C07284=1036.536,347.439,372.467,172.361,44.359,158.643
C07285=1036.529,347.192,372.505,172.355,44.357,158.642
C07286=1036.521,346.945,372.542,172.350,44.354,158.641
C07287=1036.513,346.698,372.579,172.344,44.352,158.640
C07288=1036.505,346.451,372.616,172.339,44.349,158.638
C07289=1036.498,346.204,372.654,172.332,44.347,158.637
C07290=1036.491,345.956,372.691,172.327,44.345,158.636
C07291=1036.483,345.710,372.728,172.322,44.343,158.635
C07292=1036.475,345.462,372.766,172.316,44.340,158.634
C07293=1036.467,345.215,372.803,172.310,44.338,158.633
C07294=1036.460,344.968,372.841,172.305,44.336,158.632
C07295=1036.452,344.720,372.877,172.299,44.333,158.631
C07296=1036.445,344.473,372.914,172.294,44.331,158.630
C07297=1036.437,344.226,372.951,172.289,44.329,158.629
C07298=1036.430,343.979,372.989,172.282,44.326,158.628
C07299=1036.422,343.732,373.025,172.277,44.324,158.627
C07300=1036.415,343.485,373.063,172.272,44.322,158.626
C07301=1036.407,343.238,373.099,172.266,44.320,158.625
C07302=1036.400,342.991,373.136,172.261,44.317,158.623
C07303=1036.392,342.744,373.173,172.256,44.315,158.622
C07304=1036.385,342.497,373.210,172.249,44.313,158.621
C07305=1036.378,342.249,373.247,172.244,44.310,158.620
C07306=1036.370,342.002,373.284,172.239,44.308,158.619
C07307=1036.363,341.755,373.320,172.233,44.306,158.618
C07308=1036.355,341.508,373.358,172.228,44.303,158.617
C07309=1036.348,341.260,373.394,172.223,44.301,158.616
C07310=1036.340,341.013,373.431,172.218,44.299,158.615
C07311=1036.333,340.766,373.468,172.211,44.297,158.614
C07312=1036.325,340.518,373.504,172.206,44.295,158.613
C07313=1036.318,340.272,373.541,172.201,44.293,158.612
C07314=1036.310,340.025,373.577,172.196,44.291,158.611
C07315=1036.303,339.777,373.614,172.190,44.288,158.610
C07316=1036.295,339.530,373.651,172.185,44.286,158.609
C07317=1036.287,339.283,373.687,172.180,44.284,158.608
C07318=1036.280,339.035,373.723,172.175,44.282,158.607
C07319=1036.273,338.788,373.759,172.168,44.280,158.606
C07320=1036.265,338.541,373.796,172.163,44.278,158.605
C07321=1036.258,338.294,373.833,172.158,44.275,158.604
C07322=1036.250,338.046,373.869,172.153,44.273,158.603
C07323=1036.243,337.800,373.905,172.148,44.272,158.602
C07324=1036.236,337.552,373.941,172.142,44.270,158.601
C07325=1036.228,337.304,373.978,172.137,44.267,158.600
C07326=1036.221,337.057,374.014,172.132,44.265,158.599
C07327=1036.214,336.810,374.050,172.127,44.263,158.598
C07328=1036.206,336.563,374.087,172.121,44.261,158.597
C07329=1036.199,336.316,374.124,172.116,44.259,158.597
C07330=1036.192,336.069,374.159,172.111,44.257,158.596
C07331=1036.184,335.822,374.196,172.106,44.255,158.595
C07332=1036.176,335.574,374.232,172.101,44.253,158.594
C07333=1036.165,335.199,374.287,172.093,44.250,158.592
C07334=1036.154,334.823,374.341,172.085,44.247,158.591
C07335=1036.143,334.447,374.396,172.077,44.244,158.589
C07336=1036.132,334.071,374.450,172.070,44.241,158.588
C07337=1036.125,333.824,374.487,172.064,44.238,158.587
C07338=1036.118,333.577,374.522,172.059,44.237,158.586
C07339=1036.110,333.330,374.559,172.054,44.235,158.585
C07340=1036.103,333.082,374.594,172.049,44.233,158.584
C07341=1036.095,332.835,374.630,172.044,44.231,158.583
C07342=1036.088,332.588,374.666,172.039,44.229,158.583
C07343=1036.081,332.340,374.701,172.034,44.227,158.582
C07344=1036.073,332.093,374.738,172.029,44.226,158.581
C07345=1036.066,331.846,374.773,172.023,44.223,158.580
C07346=1036.058,331.598,374.808,172.018,44.222,158.579
C07347=1036.051,331.351,374.844,172.013,44.220,158.578
C07348=1036.044,331.103,374.880,172.008,44.218,158.577
C07349=1036.037,330.857,374.916,172.003,44.216,158.576
C07350=1036.029,330.609,374.951,171.998,44.214,158.575
C07351=1036.022,330.362,374.987,171.993,44.213,158.574
C07352=1036.015,330.114,375.022,171.988,44.210,158.573
C07353=1036.008,329.867,375.058,171.983,44.209,158.573
C07354=1036.000,329.619,375.094,171.978,44.207,158.572
C07355=1035.993,329.372,375.130,171.973,44.205,158.571
C07356=1035.986,329.124,375.165,171.968,44.203,158.570
C07357=1035.979,328.877,375.201,171.963,44.202,158.569
C07358=1035.972,328.630,375.236,171.958,44.199,158.568
C07359=1035.965,328.382,375.272,171.953,44.198,158.567
C07360=1035.957,328.136,375.307,171.948,44.196,158.567
C07361=1035.950,327.888,375.342,171.943,44.195,158.566
C07362=1035.942,327.640,375.377,171.938,44.193,158.565
C07363=1035.935,327.392,375.412,171.933,44.191,158.564
C07364=1035.927,327.145,375.447,171.928,44.189,158.563
C07365=1035.920,326.898,375.482,171.924,44.187,158.562
C07366=1035.912,326.651,375.518,171.919,44.186,158.562
C07367=1035.905,326.403,375.553,171.914,44.184,158.561
C07368=1035.897,326.156,375.588,171.909,44.183,158.560
C07369=1035.890,325.908,375.623,171.904,44.181,158.559
C07370=1035.883,325.661,375.657,171.899,44.179,158.558
C07371=1035.875,325.413,375.693,171.894,44.178,158.557
C07372=1035.868,325.166,375.727,171.890,44.176,158.557
C07373=1035.861,324.919,375.763,171.885,44.174,158.556
C07374=1035.853,324.671,375.798,171.880,44.173,158.555
C07375=1035.846,324.424,375.833,171.875,44.171,158.554
C07376=1035.839,324.177,375.867,171.870,44.169,158.553
C07377=1035.831,323.929,375.903,171.865,44.168,158.553
C07378=1035.824,323.682,375.937,171.860,44.166,158.552
C07379=1035.817,323.434,375.972,171.856,44.164,158.551
C07380=1035.810,323.186,376.006,171.851,44.163,158.550
C07381=1035.803,322.938,376.042,171.846,44.161,158.549
C07382=1035.795,322.691,376.076,171.841,44.160,158.549
C07383=1035.788,322.444,376.111,171.836,44.159,158.548
C07384=1035.781,322.197,376.146,171.832,44.157,158.547
C07385=1035.774,321.950,376.181,171.827,44.155,158.546
C07386=1035.766,321.701,376.215,171.822,44.153,158.545
C07387=1035.759,321.454,376.250,171.817,44.152,158.545
C07388=1035.752,321.207,376.285,171.813,44.150,158.544
C07389=1035.741,320.826,376.339,171.806,44.148,158.543
C07390=1035.730,320.447,376.391,171.799,44.146,158.541
C07391=1035.719,320.066,376.444,171.791,44.143,158.540
C07392=1035.709,319.685,376.498,171.785,44.141,158.539
C07393=1035.701,319.438,376.532,171.780,44.139,158.538
C07394=1035.694,319.191,376.566,171.775,44.138,158.538
C07395=1035.687,318.943,376.601,171.770,44.137,158.537
C07396=1035.680,318.696,376.636,171.766,44.135,158.536
C07397=1035.673,318.448,376.670,171.761,44.133,158.535
C07398=1035.666,318.201,376.705,171.756,44.132,158.534
C07399=1035.659,317.953,376.739,171.752,44.130,158.534
C07400=1035.652,317.706,376.774,171.747,44.129,158.533
C07401=1035.645,317.458,376.808,171.742,44.128,158.532
C07402=1035.638,317.211,376.843,171.738,44.126,158.531
C07403=1035.631,316.963,376.877,171.733,44.124,158.531
C07404=1035.624,316.716,376.912,171.729,44.123,158.530
C07405=1035.617,316.468,376.946,171.725,44.121,158.529
C07406=1035.610,316.221,376.981,171.720,44.120,158.528
C07407=1035.603,315.973,377.015,171.715,44.119,158.528
C07408=1035.596,315.725,377.049,171.711,44.117,158.527
C07409=1035.589,315.478,377.083,171.706,44.116,158.526
C07410=1035.581,315.231,377.117,171.701,44.114,158.525
C07411=1035.575,314.983,377.152,171.697,44.112,158.525
C07412=1035.567,314.736,377.186,171.692,44.111,158.524
C07413=1035.562,314.488,377.220,171.687,44.110,158.523
C07414=1035.554,314.241,377.254,171.684,44.108,158.523
C07415=1035.548,313.993,377.289,171.679,44.107,158.522
C07416=1035.540,313.746,377.323,171.675,44.106,158.521
C07417=1035.533,313.498,377.357,171.670,44.104,158.520
C07418=1035.527,313.250,377.391,171.665,44.103,158.520
C07419=1035.520,313.004,377.426,171.661,44.101,158.519
C07420=1035.513,312.756,377.460,171.657,44.100,158.518
C07421=1035.506,312.508,377.494,171.653,44.098,158.517
C07422=1035.499,312.260,377.528,171.648,44.097,158.517
C07423=1035.493,312.012,377.562,171.643,44.096,158.516
C07424=1035.486,311.765,377.595,171.639,44.094,158.515
C07425=1035.479,311.518,377.629,171.634,44.093,158.515
C07426=1035.472,311.270,377.663,171.630,44.091,158.514
C07427=1035.464,311.022,377.697,171.626,44.090,158.513
C07428=1035.457,310.775,377.731,171.621,44.089,158.513
C07429=1035.450,310.527,377.765,171.617,44.088,158.512
C07430=1035.443,310.280,377.797,171.612,44.087,158.511
C07431=1035.435,310.033,377.831,171.608,44.085,158.511
C07432=1035.428,309.785,377.865,171.604,44.084,158.510
C07433=1035.421,309.537,377.898,171.599,44.083,158.509
C07434=1035.414,309.289,377.932,171.595,44.082,158.509
C07435=1035.407,309.042,377.965,171.590,44.080,158.508
C07436=1035.400,308.795,377.999,171.586,44.079,158.507
C07437=1035.393,308.546,378.032,171.582,44.078,158.507
C07438=1035.385,308.299,378.066,171.577,44.077,158.506
C07439=1035.379,308.052,378.099,171.573,44.076,158.505
C07440=1035.371,307.804,378.132,171.568,44.075,158.505
C07441=1035.364,307.556,378.165,171.565,44.074,158.504
C07442=1035.357,307.308,378.199,171.560,44.073,158.503
C07443=1035.350,307.061,378.233,171.556,44.071,158.503
C07444=1035.343,306.813,378.266,171.551,44.070,158.502
C07445=1035.332,306.438,378.316,171.545,44.068,158.501
C07446=1035.322,306.063,378.367,171.538,44.066,158.500
C07447=1035.311,305.687,378.418,171.532,44.065,158.499
C07448=1035.300,305.312,378.467,171.526,44.063,158.498
C07449=1035.293,305.064,378.501,171.521,44.062,158.497
C07450=1035.286,304.816,378.534,171.517,44.061,158.497
C07451=1035.280,304.569,378.567,171.512,44.060,158.496
C07452=1035.272,304.321,378.601,171.509,44.058,158.496
C07453=1035.261,303.916,378.655,171.501,44.057,158.495
C07454=1035.250,303.511,378.709,171.494,44.055,158.493
C07455=1035.238,303.106,378.763,171.487,44.053,158.493
C07456=1035.227,302.701,378.817,171.481,44.051,158.492
C07457=1035.220,302.453,378.850,171.476,44.050,158.491
C07458=1035.213,302.205,378.883,171.473,44.049,158.490
C07459=1035.206,301.957,378.917,171.468,44.048,158.490
C07460=1035.199,301.710,378.949,171.464,44.047,158.489
C07461=1035.192,301.462,378.982,171.459,44.046,158.488
C07462=1035.186,301.215,379.016,171.456,44.045,158.488
C07463=1035.179,300.966,379.049,171.452,44.043,158.487
C07464=1035.172,300.719,379.081,171.447,44.043,158.487
C07465=1035.165,300.471,379.114,171.444,44.042,158.486
C07466=1035.158,300.224,379.147,171.439,44.041,158.485
C07467=1035.152,299.976,379.180,171.435,44.039,158.485
C07468=1035.144,299.728,379.213,171.430,44.038,158.484
C07469=1035.138,299.481,379.245,171.427,44.037,158.483
C07470=1035.131,299.232,379.278,171.423,44.036,158.483
C07471=1035.124,298.985,379.312,171.418,44.035,158.482
C07472=1035.117,298.737,379.344,171.415,44.034,158.482
C07473=1035.111,298.490,379.377,171.410,44.033,158.481
C07474=1035.104,298.242,379.410,171.406,44.032,158.481
C07475=1035.097,297.994,379.443,171.402,44.031,158.480
C07476=1035.090,297.747,379.475,171.398,44.030,158.479
C07477=1035.084,297.499,379.508,171.394,44.029,158.479
C07478=1035.077,297.251,379.541,171.390,44.028,158.478
C07479=1035.071,297.003,379.574,171.386,44.027,158.478
C07480=1035.064,296.756,379.606,171.382,44.026,158.477
C07481=1035.057,296.508,379.639,171.378,44.025,158.476
C07482=1035.051,296.260,379.672,171.374,44.024,158.476
C07483=1035.044,296.012,379.705,171.370,44.022,158.475
C07484=1035.037,295.764,379.737,171.366,44.022,158.475
C07485=1035.030,295.517,379.770,171.362,44.021,158.474
C07486=1035.024,295.269,379.803,171.358,44.019,158.473
C07487=1035.016,295.021,379.835,171.354,44.018,158.473
C07488=1035.010,294.774,379.868,171.350,44.018,158.472
C07489=1035.003,294.526,379.900,171.346,44.017,158.472
C07490=1034.996,294.278,379.933,171.341,44.016,158.471
C07491=1034.989,294.031,379.965,171.338,44.015,158.471
C07492=1034.983,293.783,379.997,171.334,44.014,158.470
C07493=1034.976,293.535,380.030,171.329,44.013,158.470
C07494=1034.969,293.287,380.062,171.326,44.013,158.469
C07495=1034.963,293.039,380.094,171.322,44.011,158.469
C07496=1034.956,292.792,380.126,171.318,44.011,158.468
C07497=1034.949,292.567,380.156,171.314,44.010,158.467
C07498=1034.943,292.343,380.185,171.311,44.009,158.467
C07499=1034.937,292.118,380.214,171.307,44.008,158.467
C07500=1034.930,291.894,380.243,171.304,44.008,158.466
C07501=1034.924,291.670,380.272,171.300,44.006,158.465
C07502=1034.918,291.446,380.301,171.296,44.006,158.465
C07503=1034.912,291.221,380.330,171.293,44.005,158.465
C07504=1034.906,290.997,380.360,171.289,44.005,158.464
C07505=1034.899,290.749,380.391,171.286,44.003,158.463
C07506=1034.892,290.501,380.424,171.282,44.003,158.463
C07507=1034.885,290.253,380.455,171.277,44.002,158.462
C07508=1034.879,290.005,380.488,171.274,44.001,158.462
C07509=1034.872,289.758,380.519,171.270,44.000,158.461
C07510=1034.865,289.510,380.551,171.267,43.999,158.461
C07511=1034.857,289.262,380.583,171.262,43.999,158.460
C07512=1034.851,289.014,380.616,171.259,43.998,158.460
C07513=1034.844,288.766,380.647,171.255,43.997,158.459
C07514=1034.838,288.518,380.679,171.250,43.996,158.459
C07515=1034.831,288.271,380.711,171.247,43.996,158.458
C07516=1034.823,288.022,380.743,171.243,43.994,158.458
C07517=1034.816,287.775,380.775,171.240,43.994,158.457
C07518=1034.810,287.527,380.807,171.235,43.993,158.457
C07519=1034.804,287.279,380.838,171.231,43.992,158.456
C07520=1034.797,287.032,380.870,171.228,43.991,158.456
C07521=1034.790,286.784,380.902,171.224,43.991,158.455
C07522=1034.783,286.536,380.933,171.220,43.990,158.455
C07523=1034.776,286.288,380.965,171.216,43.989,158.454
C07524=1034.769,286.040,380.997,171.213,43.988,158.454
C07525=1034.762,285.792,381.029,171.209,43.988,158.453
C07526=1034.755,285.544,381.060,171.205,43.987,158.453
C07527=1034.749,285.296,381.092,171.201,43.986,158.452
C07528=1034.742,285.048,381.123,171.197,43.985,158.452
C07529=1034.735,284.801,381.154,171.194,43.985,158.451
C07530=1034.728,284.553,381.187,171.189,43.984,158.451
C07531=1034.721,284.305,381.218,171.186,43.984,158.450
C07532=1034.714,284.057,381.250,171.182,43.983,158.450
C07533=1034.707,283.809,381.281,171.179,43.982,158.449
C07534=1034.701,283.561,381.313,171.174,43.981,158.449
C07535=1034.694,283.313,381.344,171.171,43.981,158.448
C07536=1034.687,283.065,381.376,171.167,43.980,158.448
C07537=1034.680,282.817,381.407,171.164,43.979,158.447
C07538=1034.674,282.569,381.438,171.160,43.979,158.447
C07539=1034.667,282.321,381.470,171.156,43.978,158.447
C07540=1034.660,282.074,381.501,171.152,43.978,158.446
C07541=1034.654,281.826,381.533,171.148,43.976,158.445
C07542=1034.647,281.578,381.564,171.145,43.976,158.445
C07543=1034.640,281.330,381.596,171.141,43.975,158.445
C07544=1034.633,281.082,381.627,171.137,43.975,158.444
C07545=1034.627,280.834,381.658,171.133,43.974,158.444
C07546=1034.619,280.586,381.689,171.130,43.973,158.443
C07547=1034.612,280.339,381.721,171.126,43.973,158.443
C07548=1034.606,280.090,381.751,171.123,43.972,158.442
C07549=1034.599,279.842,381.783,171.119,43.972,158.442
C07550=1034.593,279.594,381.814,171.115,43.971,158.441
C07551=1034.586,279.346,381.846,171.111,43.970,158.441
C07552=1034.579,279.098,381.877,171.108,43.970,158.440
C07553=1034.573,278.851,381.908,171.104,43.969,158.440
C07554=1034.567,278.603,381.939,171.101,43.968,158.440
C07555=1034.560,278.355,381.970,171.097,43.968,158.439
C07556=1034.553,278.107,382.002,171.094,43.967,158.439
C07557=1034.544,277.761,382.045,171.088,43.966,158.438
C07558=1034.534,277.414,382.088,171.083,43.965,158.437
C07559=1034.524,277.067,382.131,171.078,43.965,158.437
C07560=1034.515,276.721,382.175,171.073,43.964,158.436
C07561=1034.508,276.473,382.206,171.070,43.963,158.436
C07562=1034.501,276.224,382.237,171.066,43.963,158.435
C07563=1034.494,275.977,382.268,171.063,43.962,158.435
C07564=1034.488,275.728,382.299,171.058,43.962,158.434
C07565=1034.481,275.480,382.330,171.055,43.961,158.434
C07566=1034.475,275.233,382.360,171.051,43.961,158.434
C07567=1034.468,274.985,382.391,171.048,43.960,158.433
C07568=1034.461,274.737,382.423,171.044,43.960,158.433
C07569=1034.454,274.489,382.453,171.041,43.959,158.432
C07570=1034.447,274.241,382.484,171.037,43.958,158.432
C07571=1034.441,273.992,382.515,171.034,43.958,158.431
C07572=1034.435,273.745,382.545,171.030,43.957,158.431
C07573=1034.427,273.497,382.576,171.027,43.957,158.431
C07574=1034.421,273.249,382.607,171.023,43.956,158.430
C07575=1034.413,273.001,382.638,171.019,43.956,158.430
C07576=1034.407,272.752,382.668,171.016,43.955,158.429
C07577=1034.400,272.505,382.700,171.012,43.955,158.429
C07578=1034.394,272.257,382.729,171.009,43.954,158.428
C07579=1034.387,272.009,382.760,171.005,43.954,158.428
C07580=1034.380,271.761,382.791,171.002,43.953,158.428
C07581=1034.373,271.512,382.822,170.998,43.953,158.427
C07582=1034.368,271.265,382.852,170.995,43.953,158.427
C07583=1034.360,271.017,382.883,170.992,43.952,158.426
C07584=1034.354,270.768,382.914,170.988,43.951,158.426
C07585=1034.347,270.520,382.944,170.985,43.951,158.425
C07586=1034.341,270.272,382.974,170.981,43.951,158.425
C07587=1034.333,270.025,383.005,170.978,43.950,158.425
C07588=1034.326,269.777,383.035,170.973,43.949,158.424
C07589=1034.320,269.528,383.066,170.970,43.949,158.424
C07590=1034.313,269.281,383.096,170.967,43.949,158.423
C07591=1034.307,269.032,383.126,170.963,43.948,158.423
C07592=1034.299,268.784,383.157,170.960,43.948,158.423
C07593=1034.293,268.536,383.188,170.956,43.947,158.422
C07594=1034.286,268.288,383.218,170.953,43.947,158.422
C07595=1034.279,268.040,383.248,170.950,43.947,158.422
C07596=1034.273,267.792,383.278,170.946,43.946,158.421
C07597=1034.266,267.544,383.308,170.943,43.945,158.421
C07598=1034.260,267.296,383.339,170.939,43.945,158.420
C07599=1034.253,267.047,383.369,170.936,43.945,158.420
C07600=1034.246,266.800,383.400,170.932,43.945,158.420
C07601=1034.239,266.552,383.430,170.929,43.944,158.419
C07602=1034.232,266.304,383.460,170.926,43.943,158.419
C07603=1034.225,266.056,383.490,170.922,43.943,158.418
C07604=1034.219,265.807,383.520,170.919,43.943,158.418
C07605=1034.212,265.559,383.550,170.915,43.943,158.418
C07606=1034.205,265.311,383.580,170.912,43.942,158.417
C07607=1034.199,265.063,383.610,170.909,43.942,158.417
C07608=1034.192,264.815,383.641,170.905,43.941,158.416
C07609=1034.186,264.567,383.671,170.902,43.941,158.416
C07610=1034.178,264.319,383.701,170.898,43.941,158.416
C07611=1034.172,264.070,383.731,170.895,43.941,158.415
C07612=1034.165,263.823,383.761,170.892,43.940,158.415
C07613=1034.156,263.481,383.803,170.887,43.939,158.415
C07614=1034.147,263.139,383.844,170.883,43.939,158.414
C07615=1034.138,262.798,383.885,170.878,43.939,158.414
C07616=1034.129,262.455,383.926,170.874,43.938,158.413
C07617=1034.122,262.207,383.956,170.870,43.937,158.413
C07618=1034.115,261.959,383.986,170.867,43.937,158.412
C07619=1034.109,261.711,384.017,170.863,43.937,158.412
C07620=1034.102,261.463,384.047,170.860,43.937,158.412
C07621=1034.095,261.215,384.076,170.857,43.936,158.411
C07622=1034.088,260.966,384.106,170.853,43.936,158.411
C07623=1034.081,260.718,384.135,170.850,43.936,158.411
C07624=1034.074,260.470,384.165,170.847,43.935,158.410
C07625=1034.067,260.222,384.195,170.843,43.935,158.410
C07626=1034.061,259.974,384.224,170.840,43.935,158.409
C07627=1034.053,259.726,384.254,170.837,43.935,158.409
C07628=1034.047,259.478,384.283,170.833,43.935,158.409
C07629=1034.040,259.229,384.313,170.830,43.935,158.408
C07630=1034.033,258.981,384.342,170.827,43.934,158.408
C07631=1034.026,258.733,384.372,170.823,43.934,158.408
C07632=1034.019,258.484,384.401,170.820,43.934,158.407
C07633=1034.013,258.237,384.431,170.817,43.934,158.407
C07634=1034.006,257.988,384.460,170.813,43.933,158.407
C07635=1033.999,257.741,384.490,170.810,43.933,158.406
C07636=1033.992,257.492,384.519,170.807,43.933,158.406
C07637=1033.986,257.244,384.549,170.803,43.933,158.406
C07638=1033.979,256.995,384.579,170.800,43.932,158.405
C07639=1033.972,256.748,384.608,170.797,43.932,158.405
C07640=1033.965,256.499,384.637,170.793,43.932,158.405
C07641=1033.958,256.251,384.666,170.790,43.932,158.404
C07642=1033.951,256.003,384.696,170.788,43.931,158.404
C07643=1033.945,255.755,384.725,170.784,43.931,158.404
C07644=1033.938,255.507,384.755,170.781,43.931,158.404
C07645=1033.932,255.259,384.784,170.778,43.931,158.403
C07646=1033.924,255.010,384.813,170.774,43.931,158.403
C07647=1033.917,254.763,384.843,170.771,43.931,158.402
C07648=1033.911,254.514,384.872,170.768,43.930,158.402
C07649=1033.904,254.266,384.901,170.765,43.930,158.402
C07650=1033.898,254.018,384.931,170.761,43.930,158.401
C07651=1033.891,253.769,384.961,170.758,43.930,158.401
C07652=1033.884,253.521,384.989,170.755,43.930,158.401
C07653=1033.877,253.273,385.018,170.752,43.929,158.401
C07654=1033.871,253.025,385.048,170.749,43.929,158.400
C07655=1033.864,252.776,385.078,170.746,43.929,158.400
C07656=1033.857,252.528,385.107,170.742,43.929,158.400
C07657=1033.851,252.280,385.136,170.739,43.929,158.399
C07658=1033.843,252.032,385.165,170.736,43.929,158.399
C07659=1033.837,251.784,385.194,170.732,43.928,158.399
C07660=1033.831,251.536,385.223,170.730,43.928,158.398
C07661=1033.824,251.287,385.253,170.727,43.928,158.398
C07662=1033.818,251.039,385.282,170.723,43.928,158.398
C07663=1033.811,250.791,385.312,170.720,43.928,158.397
C07664=1033.804,250.543,385.340,170.717,43.927,158.397
C07665=1033.797,250.295,385.369,170.713,43.927,158.397
C07666=1033.791,250.047,385.398,170.710,43.927,158.396
C07667=1033.784,249.798,385.428,170.708,43.927,158.396
C07668=1033.778,249.550,385.457,170.705,43.927,158.396
C07669=1033.768,249.207,385.498,170.700,43.926,158.395
C07670=1033.760,248.864,385.538,170.696,43.926,158.395
C07671=1033.750,248.520,385.578,170.691,43.926,158.395
C07672=1033.741,248.177,385.618,170.687,43.925,158.394
C07673=1033.735,247.929,385.647,170.684,43.925,158.394
C07674=1033.728,247.680,385.676,170.681,43.925,158.394
C07675=1033.722,247.432,385.705,170.678,43.925,158.393
C07676=1033.715,247.184,385.734,170.675,43.925,158.393
C07677=1033.709,246.936,385.763,170.671,43.924,158.392
C07678=1033.702,246.687,385.792,170.668,43.924,158.392
C07679=1033.696,246.439,385.821,170.666,43.924,158.392
C07680=1033.689,246.191,385.850,170.663,43.924,158.392
C07681=1033.682,245.943,385.879,170.659,43.924,158.391
C07682=1033.676,245.694,385.908,170.656,43.924,158.391
C07683=1033.669,245.446,385.937,170.654,43.924,158.391
C07684=1033.663,245.198,385.966,170.650,43.923,158.390
C07685=1033.657,244.950,385.995,170.647,43.923,158.390
C07686=1033.650,244.702,386.024,170.644,43.923,158.390
C07687=1033.643,244.452,386.052,170.641,43.923,158.390
C07688=1033.637,244.204,386.081,170.638,43.923,158.389
C07689=1033.630,243.956,386.110,170.635,43.923,158.389
C07690=1033.624,243.708,386.139,170.632,43.923,158.389
C07691=1033.617,243.461,386.167,170.628,43.923,158.388
C07692=1033.610,243.211,386.196,170.626,43.922,158.388
C07693=1033.603,242.963,386.224,170.623,43.922,158.388
C07694=1033.597,242.715,386.253,170.620,43.922,158.388
C07695=1033.590,242.467,386.282,170.616,43.922,158.387
C07696=1033.584,242.219,386.310,170.614,43.922,158.387
C07697=1033.577,241.970,386.339,170.611,43.922,158.387
C07698=1033.570,241.722,386.368,170.608,43.922,158.386
C07699=1033.564,241.473,386.396,170.604,43.922,158.386
C07700=1033.557,241.225,386.425,170.602,43.922,158.386
C07701=1033.550,240.977,386.453,170.599,43.922,158.386
C07702=1033.544,240.729,386.482,170.596,43.922,158.385
C07703=1033.537,240.481,386.510,170.592,43.921,158.385
C07704=1033.531,240.232,386.539,170.590,43.921,158.385
C07705=1033.524,239.984,386.567,170.587,43.921,158.384
C07706=1033.517,239.736,386.596,170.583,43.921,158.384
C07707=1033.511,239.487,386.624,170.580,43.922,158.384
C07708=1033.504,239.239,386.652,170.578,43.922,158.384
C07709=1033.497,238.991,386.680,170.575,43.921,158.383
C07710=1033.490,238.742,386.710,170.572,43.921,158.383
C07711=1033.484,238.494,386.737,170.568,43.921,158.383
C07712=1033.477,238.246,386.766,170.566,43.921,158.383
C07713=1033.470,237.997,386.793,170.563,43.921,158.382
C07714=1033.464,237.749,386.823,170.560,43.921,158.382
C07715=1033.457,237.501,386.850,170.557,43.922,158.382
C07716=1033.450,237.253,386.879,170.554,43.921,158.382
C07717=1033.443,237.004,386.906,170.551,43.921,158.381
C07718=1033.438,236.756,386.935,170.548,43.921,158.381
C07719=1033.430,236.507,386.964,170.544,43.921,158.381
C07720=1033.423,236.259,386.991,170.542,43.921,158.381
C07721=1033.416,236.011,387.020,170.539,43.922,158.380
C07722=1033.410,235.762,387.047,170.536,43.922,158.380
C07723=1033.404,235.514,387.076,170.534,43.921,158.380
C07724=1033.397,235.266,387.104,170.530,43.921,158.380
C07725=1033.387,234.916,387.144,170.526,43.921,158.379
C07726=1033.378,234.568,387.183,170.522,43.922,158.379
C07727=1033.368,234.218,387.222,170.519,43.922,158.379
C07728=1033.359,233.869,387.262,170.514,43.922,158.378
C07729=1033.352,233.620,387.290,170.511,43.922,158.378
C07730=1033.346,233.372,387.318,170.508,43.922,158.378
C07731=1033.339,233.123,387.346,170.506,43.921,158.377
C07732=1033.332,232.875,387.374,170.502,43.921,158.377
C07733=1033.326,232.627,387.402,170.499,43.922,158.377
C07734=1033.319,232.378,387.430,170.497,43.922,158.377
C07735=1033.313,232.130,387.458,170.494,43.922,158.376
C07736=1033.306,231.882,387.487,170.490,43.922,158.376
C07737=1033.299,231.633,387.514,170.488,43.922,158.376
C07738=1033.293,231.385,387.542,170.485,43.922,158.376
C07739=1033.286,231.137,387.570,170.482,43.922,158.376
C07740=1033.279,230.888,387.598,170.480,43.922,158.375
C07741=1033.273,230.640,387.625,170.477,43.922,158.375
C07742=1033.267,230.392,387.653,170.473,43.922,158.375
C07743=1033.260,230.144,387.681,170.471,43.922,158.375
C07744=1033.253,229.896,387.709,170.468,43.922,158.374
C07745=1033.246,229.647,387.737,170.465,43.922,158.374
C07746=1033.240,229.399,387.764,170.463,43.922,158.374
C07747=1033.233,229.150,387.792,170.459,43.922,158.374
C07748=1033.227,228.902,387.820,170.456,43.923,158.373
C07749=1033.220,228.653,387.848,170.454,43.923,158.373
C07750=1033.214,228.405,387.876,170.451,43.923,158.373
C07751=1033.207,228.156,387.904,170.448,43.922,158.373
C07752=1033.200,227.908,387.931,170.445,43.923,158.373
C07753=1033.193,227.660,387.958,170.442,43.923,158.372
C07754=1033.186,227.411,387.986,170.440,43.923,158.372
C07755=1033.179,227.163,388.014,170.437,43.923,158.372
C07756=1033.173,226.914,388.042,170.434,43.923,158.372
C07757=1033.166,226.666,388.069,170.432,43.923,158.371
C07758=1033.160,226.417,388.096,170.428,43.923,158.371
C07759=1033.153,226.169,388.123,170.425,43.923,158.371
C07760=1033.146,225.921,388.151,170.423,43.924,158.371
C07761=1033.140,225.673,388.179,170.420,43.924,158.371
C07762=1033.133,225.424,388.206,170.418,43.924,158.370
C07763=1033.126,225.176,388.234,170.414,43.924,158.370
C07764=1033.119,224.928,388.261,170.411,43.925,158.370
C07765=1033.112,224.679,388.288,170.409,43.924,158.370
C07766=1033.106,224.430,388.316,170.406,43.924,158.369
C07767=1033.099,224.182,388.344,170.403,43.925,158.369
C07768=1033.092,223.933,388.371,170.401,43.925,158.369
C07769=1033.086,223.686,388.398,170.398,43.925,158.369
C07770=1033.079,223.437,388.425,170.395,43.925,158.369
C07771=1033.072,223.188,388.453,170.392,43.925,158.368
C07772=1033.066,222.940,388.481,170.389,43.926,158.368
C07773=1033.059,222.691,388.508,170.387,43.925,158.368
C07774=1033.052,222.443,388.535,170.384,43.926,158.368
C07775=1033.045,222.194,388.562,170.381,43.926,158.368
C07776=1033.039,221.946,388.590,170.378,43.926,158.367
C07777=1033.033,221.697,388.617,170.375,43.926,158.367
C07778=1033.025,221.449,388.644,170.373,43.926,158.367
C07779=1033.019,221.201,388.672,170.370,43.927,158.367
C07780=1033.012,220.952,388.699,170.368,43.926,158.367
C07781=1033.003,220.596,388.739,170.363,43.926,158.366
C07782=1032.993,220.239,388.778,170.359,43.927,158.366
C07783=1032.984,219.883,388.817,170.356,43.927,158.366
C07784=1032.975,219.526,388.856,170.352,43.927,158.365
C07785=1032.968,219.277,388.882,170.348,43.927,158.365
C07786=1032.961,219.028,388.910,170.346,43.928,158.365
C07787=1032.954,218.780,388.936,170.343,43.928,158.365
C07788=1032.947,218.531,388.964,170.341,43.928,158.365
C07789=1032.941,218.283,388.990,170.338,43.929,158.364
C07790=1032.934,218.035,389.018,170.336,43.928,158.364
C07791=1032.927,217.786,389.044,170.333,43.929,158.364
C07792=1032.920,217.538,389.072,170.330,43.929,158.364
C07793=1032.913,217.289,389.098,170.328,43.929,158.364
C07794=1032.907,217.041,389.126,170.324,43.929,158.363
C07795=1032.900,216.792,389.152,170.322,43.930,158.363
C07796=1032.893,216.544,389.180,170.319,43.930,158.363
C07797=1032.886,216.295,389.206,170.317,43.930,158.363
C07798=1032.880,216.047,389.234,170.314,43.931,158.363
C07799=1032.873,215.799,389.260,170.312,43.930,158.363
C07800=1032.867,215.550,389.287,170.309,43.931,158.362
C07801=1032.859,215.301,389.314,170.306,43.931,158.362
C07802=1032.854,215.053,389.341,170.303,43.931,158.362
C07803=1032.846,214.805,389.368,170.300,43.932,158.362
C07804=1032.840,214.556,389.395,170.298,43.932,158.362
C07805=1032.833,214.308,389.421,170.295,43.932,158.361
C07806=1032.827,214.059,389.449,170.293,43.932,158.361
C07807=1032.819,213.811,389.475,170.290,43.933,158.361
C07808=1032.813,213.562,389.502,170.287,43.932,158.361
C07809=1032.806,213.314,389.529,170.284,43.933,158.361
C07810=1032.800,213.065,389.556,170.282,43.933,158.360
C07811=1032.793,212.816,389.582,170.279,43.933,158.360
C07812=1032.787,212.569,389.610,170.277,43.934,158.360
C07813=1032.780,212.320,389.636,170.274,43.934,158.360
C07814=1032.773,212.071,389.663,170.272,43.934,158.360
C07815=1032.767,211.823,389.689,170.268,43.934,158.360
C07816=1032.760,211.574,389.717,170.266,43.934,158.359
C07817=1032.753,211.326,389.743,170.263,43.934,158.359
C07818=1032.747,211.077,389.770,170.261,43.935,158.359
C07819=1032.740,210.828,389.797,170.258,43.935,158.359
C07820=1032.733,210.580,389.823,170.256,43.935,158.359
C07821=1032.727,210.332,389.850,170.253,43.936,158.359
C07822=1032.720,210.083,389.877,170.251,43.936,158.358
C07823=1032.713,209.835,389.903,170.248,43.936,158.358
C07824=1032.707,209.586,389.930,170.246,43.936,158.358
C07825=1032.700,209.337,389.956,170.242,43.937,158.358
C07826=1032.693,209.089,389.982,170.240,43.937,158.358
C07827=1032.687,208.840,390.009,170.237,43.937,158.358
C07828=1032.680,208.593,390.036,170.235,43.938,158.357
C07829=1032.673,208.344,390.062,170.233,43.937,158.357
C07830=1032.666,208.095,390.089,170.230,43.938,158.357
C07831=1032.660,207.847,390.116,170.228,43.938,158.357
C07832=1032.653,207.598,390.142,170.225,43.938,158.357
C07833=1032.646,207.350,390.168,170.223,43.939,158.357
C07834=1032.639,207.101,390.194,170.220,43.939,158.356
C07835=1032.632,206.853,390.221,170.217,43.939,158.356
C07836=1032.626,206.604,390.248,170.214,43.940,158.356
C07837=1032.617,206.253,390.284,170.211,43.940,158.356
C07838=1032.606,205.902,390.322,170.207,43.940,158.356
C07839=1032.597,205.551,390.359,170.204,43.941,158.355
C07840=1032.588,205.200,390.396,170.200,43.942,158.355
C07841=1032.562,204.151,390.501,169.861,43.837,158.304
C07842=1032.556,203.902,390.527,169.857,43.838,158.304
C07843=1032.550,203.653,390.551,169.853,43.839,158.304
C07844=1032.544,203.405,390.576,169.850,43.840,158.304
C07845=1032.537,203.157,390.601,169.846,43.842,158.304
C07846=1032.531,202.907,390.626,169.842,43.842,158.304
C07847=1032.525,202.659,390.651,169.839,43.844,158.304
C07848=1032.519,202.411,390.676,169.835,43.844,158.304
C07849=1032.514,202.161,390.701,169.832,43.846,158.304
C07850=1032.507,201.913,390.726,169.828,43.847,158.304
C07851=1032.501,201.664,390.751,169.825,43.848,158.303
C07852=1032.495,201.416,390.775,169.822,43.849,158.303
C07853=1032.489,201.167,390.800,169.817,43.850,158.303
C07854=1032.483,200.918,390.825,169.815,43.851,158.303
C07855=1032.477,200.669,390.850,169.811,43.852,158.303
C07856=1032.472,200.421,390.875,169.808,43.853,158.303
C07857=1032.465,200.172,390.899,169.804,43.854,158.303
C07858=1032.459,199.923,390.924,169.800,43.856,158.303
C07859=1032.452,199.675,390.949,169.797,43.857,158.303
C07860=1032.446,199.426,390.973,169.794,43.858,158.303
C07861=1032.440,199.177,390.997,169.790,43.859,158.303
C07862=1032.434,198.928,391.022,169.787,43.860,158.303
C07863=1032.427,198.679,391.046,169.783,43.862,158.303
C07864=1032.422,198.431,391.071,169.780,43.863,158.303
C07865=1032.415,198.182,391.095,169.776,43.865,158.303
C07866=1032.409,197.933,391.120,169.773,43.865,158.302
C07867=1032.403,197.685,391.144,169.769,43.867,158.302
C07868=1032.397,197.436,391.169,169.765,43.868,158.302
C07869=1032.390,197.187,391.193,169.763,43.869,158.302
C07870=1032.384,196.938,391.218,169.759,43.871,158.302
C07871=1032.378,196.690,391.242,169.756,43.872,158.302
C07872=1032.372,196.441,391.267,169.752,43.873,158.302
C07873=1032.365,196.192,391.291,169.749,43.874,158.302
C07874=1032.360,195.943,391.315,169.745,43.875,158.302
C07875=1032.353,195.695,391.340,169.741,43.877,158.302
C07876=1032.348,195.446,391.364,169.739,43.878,158.302
C07877=1032.341,195.197,391.388,169.735,43.879,158.302
C07878=1032.335,194.948,391.413,169.732,43.880,158.302
C07879=1032.329,194.701,391.437,169.728,43.882,158.302
C07880=1032.323,194.451,391.462,169.725,43.882,158.302
C07881=1032.316,194.202,391.486,169.721,43.884,158.302
C07882=1032.311,193.954,391.510,169.719,43.885,158.302
C07883=1032.304,193.705,391.534,169.715,43.886,158.302
C07884=1032.299,193.456,391.558,169.712,43.888,158.302
C07885=1032.292,193.208,391.583,169.708,43.889,158.302
C07886=1032.287,192.959,391.607,169.705,43.890,158.302
C07887=1032.280,192.710,391.631,169.701,43.892,158.302
C07888=1032.274,192.461,391.656,169.699,43.893,158.302
C07889=1032.268,192.213,391.679,169.695,43.894,158.302
C07890=1032.262,191.963,391.704,169.692,43.895,158.302
C07891=1032.256,191.715,391.728,169.688,43.896,158.302
C07892=1032.250,191.466,391.752,169.685,43.898,158.302
C07893=1032.244,191.217,391.776,169.681,43.899,158.301
C07894=1032.238,190.968,391.801,169.678,43.900,158.301
C07895=1032.232,190.720,391.824,169.675,43.902,158.301
C07896=1032.226,190.471,391.849,169.672,43.903,158.301
C07897=1032.220,190.222,391.873,169.668,43.904,158.301
C07898=1032.214,189.973,391.897,169.665,43.906,158.301
C07899=1032.208,189.725,391.921,169.661,43.907,158.301
C07900=1032.202,189.476,391.945,169.658,43.908,158.301
C07901=1032.196,189.227,391.969,169.656,43.909,158.301
C07902=1032.190,188.944,391.997,169.652,43.911,158.301
C07903=1032.183,188.660,392.024,169.648,43.912,158.301
C07904=1032.176,188.376,392.051,169.644,43.914,158.301
C07905=1032.169,188.093,392.079,169.640,43.915,158.301
C07906=1032.163,187.844,392.103,169.637,43.916,158.301
C07907=1032.157,187.595,392.127,169.634,43.918,158.301
C07908=1032.151,187.346,392.152,169.631,43.919,158.301
C07909=1032.145,187.098,392.175,169.627,43.920,158.301
C07910=1032.140,186.849,392.199,169.624,43.922,158.301
C07911=1032.134,186.600,392.223,169.620,43.923,158.301
C07912=1032.127,186.351,392.246,169.618,43.924,158.301
C07913=1032.122,186.102,392.271,169.615,43.925,158.301
C07914=1032.116,185.854,392.295,169.611,43.927,158.301
C07915=1032.110,185.605,392.319,169.608,43.928,158.301
C07916=1032.104,185.355,392.342,169.604,43.930,158.301
C07917=1032.099,185.107,392.367,169.601,43.931,158.301
C07918=1032.093,184.859,392.390,169.599,43.932,158.301
C07919=1032.086,184.610,392.414,169.595,43.933,158.301
C07920=1032.081,184.361,392.438,169.592,43.935,158.301
C07921=1032.074,184.111,392.462,169.588,43.936,158.301
C07922=1032.069,183.863,392.486,169.585,43.937,158.301
C07923=1032.063,183.615,392.510,169.583,43.938,158.301
C07924=1032.058,183.366,392.534,169.579,43.940,158.301
C07925=1032.051,183.116,392.557,169.576,43.941,158.301
C07926=1032.045,182.868,392.581,169.573,43.942,158.301
C07927=1032.039,182.619,392.604,169.569,43.944,158.301
C07928=1032.033,182.370,392.628,169.566,43.945,158.301
C07929=1032.027,182.121,392.651,169.563,43.947,158.301
C07930=1032.020,181.873,392.674,169.560,43.948,158.301
C07931=1032.014,181.624,392.697,169.556,43.950,158.301
C07932=1032.007,181.375,392.721,169.554,43.952,158.301
C07933=1032.002,181.126,392.744,169.550,43.953,158.301
C07934=1031.996,180.878,392.768,169.547,43.954,158.301
C07935=1031.989,180.628,392.791,169.544,43.956,158.301
C07936=1031.983,180.380,392.815,169.541,43.958,158.301
C07937=1031.977,180.131,392.837,169.538,43.959,158.301
C07938=1031.971,179.882,392.860,169.534,43.961,158.301
C07939=1031.964,179.633,392.884,169.531,43.962,158.301
C07940=1031.959,179.384,392.907,169.528,43.963,158.301
C07941=1031.952,179.135,392.931,169.525,43.965,158.301
C07942=1031.946,178.887,392.954,169.522,43.967,158.301
C07943=1031.940,178.638,392.976,169.518,43.968,158.301
C07944=1031.933,178.389,393.000,169.516,43.970,158.302
C07945=1031.928,178.140,393.023,169.513,43.971,158.302
C07946=1031.922,177.891,393.046,169.509,43.973,158.301
C07947=1031.915,177.642,393.070,169.506,43.974,158.302
C07948=1031.909,177.394,393.093,169.503,43.976,158.302
C07949=1031.903,177.145,393.116,169.500,43.977,158.302
C07950=1031.897,176.896,393.139,169.497,43.979,158.302
C07951=1031.891,176.647,393.163,169.493,43.980,158.302
C07952=1031.885,176.398,393.186,169.491,43.982,158.302
C07953=1031.879,176.149,393.209,169.488,43.983,158.302
C07954=1031.872,175.900,393.232,169.484,43.985,158.302
C07955=1031.866,175.651,393.255,169.481,43.986,158.302
C07956=1031.860,175.403,393.278,169.478,43.988,158.302
C07957=1031.855,175.154,393.301,169.475,43.989,158.302
C07958=1031.849,174.905,393.324,169.472,43.991,158.302
C07959=1031.841,174.656,393.347,169.468,43.993,158.302
C07960=1031.836,174.407,393.370,169.466,43.994,158.302
C07961=1031.830,174.158,393.393,169.463,43.996,158.302
C07962=1031.824,173.909,393.416,169.459,43.997,158.302
C07963=1031.818,173.660,393.440,169.456,43.999,158.302
C07964=1031.811,173.412,393.462,169.454,44.000,158.302
C07965=1031.805,173.163,393.485,169.450,44.002,158.302
C07966=1031.799,172.879,393.511,169.447,44.004,158.302
C07967=1031.792,172.594,393.538,169.444,44.005,158.302
C07968=1031.785,172.311,393.564,169.440,44.007,158.302
C07969=1031.778,172.026,393.590,169.436,44.009,158.302
C07970=1031.772,171.777,393.613,169.434,44.011,158.303
C07971=1031.767,171.528,393.636,169.431,44.012,158.303
C07972=1031.760,171.280,393.659,169.427,44.014,158.303
C07973=1031.754,171.031,393.682,169.424,44.015,158.303
C07974=1031.748,170.783,393.705,169.422,44.016,158.303
C07975=1031.742,170.533,393.728,169.419,44.018,158.303
C07976=1031.736,170.284,393.751,169.415,44.020,158.303
C07977=1031.730,170.035,393.774,169.413,44.021,158.303
C07978=1031.724,169.787,393.796,169.410,44.023,158.303
C07979=1031.718,169.538,393.819,169.407,44.024,158.303
C07980=1031.713,169.289,393.842,169.403,44.026,158.303
C07981=1031.706,169.040,393.865,169.400,44.027,158.303
C07982=1031.700,168.791,393.888,169.398,44.029,158.303
C07983=1031.695,168.542,393.911,169.394,44.031,158.303
C07984=1031.689,168.294,393.934,169.391,44.032,158.303
C07985=1031.683,168.045,393.957,169.389,44.034,158.303
C07986=1031.677,167.796,393.979,169.386,44.035,158.303
C07987=1031.671,167.547,394.002,169.383,44.036,158.303
C07988=1031.665,167.298,394.025,169.379,44.038,158.303
C07989=1031.659,167.049,394.048,169.377,44.039,158.303
C07990=1031.652,166.800,394.070,169.374,44.041,158.303
C07991=1031.647,166.551,394.093,169.371,44.043,158.303
C07992=1031.641,166.302,394.116,169.367,44.044,158.303
C07993=1031.636,166.053,394.139,169.365,44.046,158.304
C07994=1031.629,165.804,394.161,169.362,44.047,158.304
C07995=1031.623,165.555,394.184,169.359,44.049,158.304
C07996=1031.618,165.306,394.207,169.357,44.050,158.304
C07997=1031.612,165.057,394.230,169.353,44.052,158.304
C07998=1031.605,164.809,394.252,169.350,44.054,158.304
C07999=1031.600,164.559,394.274,169.347,44.055,158.304
C08000=1031.594,164.310,394.297,169.345,44.057,158.304
C08001=1031.589,164.062,394.320,169.342,44.058,158.304
C08002=1031.583,163.814,394.342,169.338,44.060,158.304
C08003=1031.577,163.565,394.365,169.335,44.061,158.304
C08004=1031.571,163.316,394.388,169.333,44.063,158.304
C08005=1031.566,163.066,394.410,169.330,44.064,158.304
C08006=1031.559,162.818,394.433,169.327,44.066,158.304
C08007=1031.554,162.569,394.456,169.324,44.068,158.304
C08008=1031.548,162.320,394.479,169.321,44.069,158.304
C08009=1031.542,162.070,394.501,169.318,44.070,158.304
C08010=1031.536,161.822,394.523,169.315,44.072,158.304
C08011=1031.530,161.573,394.546,169.313,44.073,158.304
C08012=1031.525,161.324,394.569,169.310,44.075,158.305
C08013=1031.519,161.075,394.591,169.306,44.077,158.305
C08014=1031.513,160.826,394.614,169.304,44.079,158.305
C08015=1031.508,160.578,394.636,169.301,44.080,158.305
C08016=1031.502,160.328,394.658,169.298,44.081,158.305
C08017=1031.496,160.080,394.681,169.295,44.083,158.305
C08018=1031.490,159.831,394.704,169.293,44.084,158.305
C08019=1031.484,159.581,394.726,169.290,44.086,158.305
C08020=1031.478,159.333,394.748,169.286,44.087,158.305
C08021=1031.472,159.084,394.770,169.284,44.089,158.305
C08022=1031.466,158.835,394.793,169.281,44.091,158.305
C08023=1031.460,158.585,394.815,169.278,44.093,158.305
C08024=1031.453,158.337,394.837,169.276,44.094,158.305
C08025=1031.448,158.087,394.859,169.272,44.096,158.306
C08026=1031.442,157.839,394.881,169.269,44.098,158.306
C08027=1031.436,157.590,394.903,169.267,44.100,158.306
C08028=1031.430,157.341,394.926,169.264,44.101,158.306
C08029=1031.424,157.092,394.947,169.261,44.103,158.306
C08030=1031.417,156.808,394.973,169.258,44.105,158.306
C08031=1031.410,156.523,394.997,169.254,44.107,158.306
C08032=1031.403,156.238,395.023,169.251,44.109,158.306
C08033=1031.396,155.954,395.049,169.248,44.111,158.306
C08034=1031.390,155.705,395.070,169.245,44.112,158.306
C08035=1031.385,155.455,395.093,169.242,44.114,158.306
C08036=1031.379,155.207,395.115,169.240,44.116,158.307
C08037=1031.373,154.958,395.136,169.236,44.117,158.306
C08038=1031.366,154.710,395.159,169.233,44.119,158.307
C08039=1031.361,154.460,395.181,169.231,44.121,158.307
C08040=1031.354,154.211,395.202,169.228,44.122,158.307
C08041=1031.348,153.962,395.225,169.225,44.124,158.307
C08042=1031.343,153.713,395.247,169.223,44.126,158.307
C08043=1031.337,153.464,395.268,169.220,44.127,158.307
C08044=1031.331,153.215,395.290,169.216,44.130,158.307
C08045=1031.324,152.966,395.312,169.214,44.131,158.307
C08046=1031.318,152.717,395.334,169.211,44.133,158.307
C08047=1031.312,152.468,395.356,169.208,44.135,158.307
C08048=1031.307,152.220,395.377,169.206,44.136,158.308
C08049=1031.301,151.971,395.400,169.203,44.138,158.308
C08050=1031.295,151.721,395.421,169.199,44.140,158.308
C08051=1031.288,151.472,395.443,169.197,44.142,158.308
C08052=1031.282,151.223,395.465,169.194,44.144,158.308
C08053=1031.276,150.975,395.487,169.191,44.145,158.308
C08054=1031.270,150.726,395.508,169.189,44.147,158.308
C08055=1031.264,150.477,395.530,169.186,44.149,158.308
C08056=1031.259,150.227,395.552,169.184,44.151,158.308
C08057=1031.253,149.978,395.574,169.181,44.152,158.308
C08058=1031.247,149.730,395.595,169.177,44.154,158.308
C08059=1031.240,149.481,395.617,169.175,44.156,158.309
C08060=1031.234,149.232,395.639,169.172,44.157,158.309
C08061=1031.228,148.983,395.661,169.169,44.159,158.309
C08062=1031.223,148.734,395.682,169.167,44.161,158.309
C08063=1031.216,148.485,395.704,169.164,44.163,158.309
C08064=1031.210,148.236,395.725,169.161,44.164,158.309
C08065=1031.204,147.986,395.747,169.159,44.166,158.309
C08066=1031.199,147.738,395.768,169.156,44.168,158.309
C08067=1031.193,147.488,395.790,169.153,44.170,158.309
C08068=1031.187,147.239,395.812,169.150,44.171,158.309
C08069=1031.181,146.991,395.833,169.147,44.173,158.310
C08070=1031.175,146.741,395.855,169.145,44.175,158.310
C08071=1031.169,146.492,395.876,169.142,44.177,158.310
C08072=1031.163,146.243,395.898,169.139,44.179,158.310
C08073=1031.157,145.995,395.919,169.137,44.180,158.310
C08074=1031.150,145.746,395.940,169.134,44.182,158.310
C08075=1031.144,145.496,395.962,169.131,44.184,158.310
C08076=1031.138,145.247,395.984,169.128,44.186,158.310
C08077=1031.133,144.999,396.005,169.125,44.188,158.311
C08078=1031.126,144.750,396.027,169.123,44.190,158.311
C08079=1031.120,144.500,396.048,169.120,44.192,158.311
C08080=1031.115,144.252,396.070,169.117,44.193,158.311
C08081=1031.108,144.003,396.091,169.115,44.195,158.311
C08082=1031.102,143.754,396.112,169.112,44.197,158.311
C08083=1031.096,143.505,396.133,169.109,44.199,158.311
C08084=1031.090,143.255,396.154,169.107,44.200,158.311
C08085=1031.084,143.006,396.176,169.103,44.203,158.311
C08086=1031.078,142.758,396.197,169.100,44.204,158.311
C08087=1031.072,142.508,396.219,169.098,44.206,158.312
C08088=1031.065,142.260,396.240,169.095,44.208,158.312
C08089=1031.060,142.011,396.261,169.093,44.210,158.312
C08090=1031.054,141.761,396.282,169.090,44.211,158.312
C08091=1031.048,141.512,396.304,169.088,44.213,158.312
C08092=1031.042,141.264,396.325,169.085,44.215,158.312
C08093=1031.036,141.014,396.347,169.082,44.216,158.312
C08094=1031.029,140.730,396.371,169.079,44.219,158.312
C08095=1031.022,140.445,396.394,169.076,44.220,158.313
C08096=1031.016,140.160,396.419,169.073,44.223,158.313
C08097=1031.008,139.875,396.444,169.070,44.225,158.313
C08098=1031.003,139.625,396.465,169.067,44.226,158.313
C08099=1030.997,139.377,396.486,169.065,44.228,158.313
C08100=1030.991,139.128,396.508,169.062,44.230,158.313
C08101=1030.985,138.879,396.528,169.059,44.232,158.313
C08102=1030.979,138.630,396.549,169.057,44.234,158.314
C08103=1030.973,138.380,396.571,169.054,44.236,158.314
C08104=1030.967,138.132,396.592,169.051,44.238,158.314
C08105=1030.960,137.882,396.612,169.048,44.240,158.314
C08106=1030.955,137.634,396.634,169.045,44.242,158.314
C08107=1030.949,137.385,396.655,169.043,44.243,158.314
C08108=1030.943,137.136,396.675,169.040,44.245,158.314
C08109=1030.937,136.887,396.697,169.038,44.247,158.314
C08110=1030.931,136.637,396.718,169.035,44.249,158.314
C08111=1030.924,136.389,396.738,169.032,44.251,158.315
C08112=1030.918,136.139,396.760,169.030,44.253,158.315
C08113=1030.913,135.890,396.781,169.027,44.255,158.315
C08114=1030.906,135.641,396.802,169.025,44.256,158.315
C08115=1030.901,135.392,396.822,169.022,44.258,158.315
C08116=1030.894,135.143,396.843,169.019,44.260,158.315
C08117=1030.888,134.893,396.864,169.017,44.262,158.315
C08118=1030.882,134.645,396.885,169.014,44.264,158.316
C08119=1030.876,134.395,396.906,169.012,44.266,158.316
C08120=1030.870,134.147,396.927,169.009,44.268,158.316
C08121=1030.864,133.897,396.947,169.006,44.269,158.316
C08122=1030.858,133.649,396.969,169.004,44.271,158.316
C08123=1030.852,133.399,396.989,169.001,44.273,158.316
C08124=1030.846,133.151,397.010,168.998,44.275,158.316
C08125=1030.840,132.901,397.031,168.995,44.277,158.316
C08126=1030.834,132.653,397.052,168.992,44.279,158.317
C08127=1030.828,132.403,397.073,168.990,44.281,158.317
C08128=1030.822,132.155,397.093,168.987,44.283,158.317
C08129=1030.816,131.905,397.114,168.985,44.285,158.317
C08130=1030.811,131.656,397.135,168.982,44.287,158.317
C08131=1030.804,131.407,397.156,168.979,44.289,158.317
C08132=1030.798,131.158,397.176,168.977,44.290,158.317
C08133=1030.792,130.909,397.198,168.974,44.292,158.318
C08134=1030.786,130.660,397.218,168.972,44.294,158.318
C08135=1030.780,130.410,397.238,168.969,44.296,158.318
C08136=1030.774,130.162,397.260,168.967,44.298,158.318
C08137=1030.768,129.912,397.280,168.964,44.300,158.318
C08138=1030.762,129.664,397.300,168.961,44.302,158.318
C08139=1030.755,129.415,397.321,168.959,44.304,158.318
C08140=1030.749,129.166,397.342,168.956,44.306,158.318
C08141=1030.743,128.916,397.362,168.954,44.308,158.319
C08142=1030.737,128.667,397.382,168.951,44.310,158.319
C08143=1030.730,128.418,397.402,168.948,44.311,158.319
C08144=1030.725,128.169,397.423,168.946,44.313,158.319
C08145=1030.718,127.920,397.444,168.943,44.315,158.319
C08146=1030.712,127.671,397.464,168.941,44.318,158.319
C08147=1030.706,127.422,397.484,168.938,44.320,158.320
C08148=1030.700,127.173,397.505,168.936,44.322,158.320
C08149=1030.694,126.924,397.525,168.933,44.324,158.320
C08150=1030.687,126.674,397.546,168.931,44.326,158.320
C08151=1030.681,126.426,397.566,168.928,44.327,158.320
C08152=1030.675,126.176,397.586,168.925,44.329,158.320
C08153=1030.669,125.927,397.606,168.923,44.331,158.320
C08154=1030.663,125.679,397.627,168.920,44.333,158.321
C08155=1030.657,125.429,397.647,168.917,44.335,158.321
C08156=1030.651,125.180,397.668,168.914,44.337,158.321
C08157=1030.645,124.931,397.688,168.912,44.339,158.321
C08158=1030.638,124.646,397.711,168.909,44.342,158.321
C08159=1030.631,124.361,397.735,168.907,44.344,158.321
C08160=1030.624,124.076,397.758,168.903,44.346,158.321
C08161=1030.617,123.791,397.782,168.901,44.348,158.322
C08162=1030.611,123.542,397.802,168.898,44.350,158.322
C08163=1030.605,123.293,397.822,168.895,44.352,158.322
C08164=1030.599,123.044,397.842,168.893,44.354,158.322
C08165=1030.592,122.794,397.862,168.890,44.356,158.322
C08166=1030.587,122.545,397.883,168.888,44.358,158.322
C08167=1030.581,122.296,397.903,168.885,44.360,158.323
C08168=1030.574,122.047,397.923,168.883,44.362,158.323
C08169=1030.568,121.798,397.943,168.880,44.364,158.323
C08170=1030.563,121.549,397.964,168.877,44.366,158.323
C08171=1030.556,121.299,397.984,168.875,44.368,158.323
C08172=1030.550,121.050,398.004,168.872,44.370,158.323
C08173=1030.544,120.802,398.024,168.870,44.371,158.323
C08174=1030.538,120.552,398.044,168.867,44.373,158.324
C08175=1030.532,120.303,398.065,168.864,44.375,158.324
C08176=1030.526,120.054,398.085,168.862,44.377,158.324
C08177=1030.520,119.805,398.105,168.860,44.380,158.324
C08178=1030.514,119.556,398.125,168.857,44.382,158.324
C08179=1030.509,119.307,398.145,168.854,44.384,158.324
C08180=1030.503,119.058,398.165,168.852,44.386,158.325
C08181=1030.496,118.808,398.186,168.849,44.387,158.325
C08182=1030.490,118.560,398.206,168.847,44.389,158.325
C08183=1030.484,118.311,398.226,168.844,44.391,158.325
C08184=1030.478,118.061,398.247,168.842,44.393,158.325
C08185=1030.472,117.812,398.267,168.839,44.395,158.325
C08186=1030.466,117.563,398.286,168.836,44.397,158.325
C08187=1030.460,117.315,398.306,168.835,44.399,158.326
C08188=1030.454,117.064,398.326,168.832,44.401,158.326
C08189=1030.449,116.815,398.347,168.830,44.403,158.326
C08190=1030.443,116.566,398.367,168.827,44.405,158.326
C08191=1030.437,116.318,398.387,168.824,44.407,158.326
C08192=1030.430,116.068,398.407,168.822,44.408,158.326
C08193=1030.424,115.819,398.427,168.819,44.410,158.326
C08194=1030.419,115.570,398.447,168.817,44.412,158.326
C08195=1030.413,115.321,398.467,168.814,44.414,158.327
C08196=1030.407,115.072,398.487,168.812,44.416,158.327
C08197=1030.401,114.822,398.507,168.809,44.418,158.327
C08198=1030.395,114.574,398.527,168.806,44.420,158.327
C08199=1030.389,114.325,398.547,168.804,44.422,158.327
C08200=1030.383,114.076,398.567,168.802,44.424,158.327
C08201=1030.378,113.826,398.587,168.800,44.426,158.328
C08202=1030.371,113.577,398.607,168.797,44.427,158.328
C08203=1030.365,113.328,398.627,168.795,44.429,158.328
C08204=1030.360,113.079,398.647,168.792,44.431,158.328
C08205=1030.354,112.829,398.667,168.789,44.433,158.328
C08206=1030.347,112.580,398.687,168.787,44.435,158.328
C08207=1030.341,112.331,398.707,168.784,44.437,158.328
C08208=1030.335,112.082,398.726,168.782,44.439,158.328
C08209=1030.329,111.833,398.746,168.779,44.441,158.329
C08210=1030.323,111.584,398.766,168.776,44.443,158.329
C08211=1030.317,111.334,398.785,168.774,44.445,158.329
C08212=1030.311,111.085,398.805,168.772,44.447,158.329
C08213=1030.305,110.837,398.825,168.769,44.449,158.329
C08214=1030.299,110.587,398.844,168.767,44.451,158.329
C08215=1030.293,110.338,398.864,168.765,44.453,158.330
C08216=1030.287,110.088,398.884,168.762,44.455,158.330
C08217=1030.281,109.839,398.904,168.760,44.457,158.330
C08218=1030.274,109.591,398.923,168.757,44.459,158.330
C08219=1030.268,109.341,398.942,168.755,44.461,158.330
C08220=1030.262,109.093,398.962,168.752,44.463,158.330
C08221=1030.256,108.842,398.982,168.750,44.465,158.331
C08222=1030.249,108.557,399.004,168.746,44.467,158.331
C08223=1030.242,108.273,399.027,168.744,44.470,158.331
C08224=1030.235,107.987,399.049,168.741,44.472,158.331
C08225=1030.228,107.702,399.071,168.738,44.475,158.331
C08226=1030.222,107.453,399.090,168.735,44.477,158.331
C08227=1030.216,107.204,399.110,168.733,44.479,158.332
C08228=1030.210,106.955,399.129,168.730,44.481,158.332
C08229=1030.203,106.706,399.149,168.729,44.483,158.332
C08230=1030.197,106.456,399.168,168.726,44.485,158.332
C08231=1030.191,106.207,399.188,168.723,44.487,158.332
C08232=1030.185,105.958,399.207,168.721,44.489,158.332
C08233=1030.179,105.709,399.227,168.718,44.491,158.333
C08234=1030.173,105.460,399.246,168.716,44.493,158.333
C08235=1030.167,105.211,399.265,168.713,44.495,158.333
C08236=1030.161,104.962,399.285,168.711,44.497,158.333
C08237=1030.155,104.713,399.304,168.708,44.499,158.333
C08238=1030.149,104.463,399.324,168.706,44.501,158.333
C08239=1030.142,104.214,399.343,168.703,44.503,158.334
C08240=1030.137,103.964,399.362,168.701,44.505,158.334
C08241=1030.131,103.716,399.382,168.698,44.507,158.334
C08242=1030.125,103.466,399.401,168.696,44.509,158.334
C08243=1030.118,103.217,399.420,168.694,44.511,158.334
C08244=1030.112,102.968,399.440,168.691,44.513,158.334
C08245=1030.107,102.719,399.459,168.689,44.515,158.335
C08246=1030.100,102.470,399.479,168.686,44.517,158.335
C08247=1030.094,102.221,399.498,168.684,44.519,158.335
C08248=1030.089,101.972,399.517,168.681,44.521,158.335
C08249=1030.083,101.722,399.536,168.679,44.523,158.335
C08250=1030.076,101.474,399.556,168.676,44.525,158.335
C08251=1030.071,101.224,399.575,168.674,44.527,158.335
C08252=1030.065,100.975,399.594,168.671,44.529,158.336
C08253=1030.058,100.726,399.614,168.670,44.531,158.336
C08254=1030.052,100.476,399.633,168.667,44.533,158.336
C08255=1030.046,100.227,399.653,168.664,44.535,158.336
C08256=1030.040,99.977,399.672,168.662,44.537,158.336
C08257=1030.034,99.729,399.691,168.659,44.539,158.336
C08258=1030.028,99.479,399.710,168.657,44.541,158.337
C08259=1030.022,99.230,399.729,168.654,44.543,158.337
C08260=1030.016,98.981,399.748,168.652,44.545,158.337
C08261=1030.009,98.732,399.767,168.649,44.548,158.337
C08262=1030.003,98.482,399.786,168.647,44.550,158.337
C08263=1029.997,98.234,399.806,168.644,44.552,158.337
C08264=1029.991,97.985,399.824,168.642,44.554,158.338
C08265=1029.985,97.735,399.843,168.640,44.556,158.338
C08266=1029.979,97.486,399.862,168.638,44.558,158.338
C08267=1029.973,97.237,399.881,168.635,44.560,158.338
C08268=1029.966,96.987,399.900,168.633,44.562,158.338
C08269=1029.961,96.738,399.919,168.630,44.564,158.339
C08270=1029.954,96.489,399.938,168.628,44.566,158.339
C08271=1029.948,96.240,399.956,168.625,44.568,158.339
C08272=1029.942,95.990,399.976,168.623,44.570,158.339
C08273=1029.935,95.742,399.995,168.620,44.572,158.339
C08274=1029.930,95.492,400.014,168.618,44.575,158.339
C08275=1029.923,95.243,400.033,168.615,44.577,158.339
C08276=1029.918,94.994,400.052,168.612,44.579,158.340
C08277=1029.911,94.745,400.071,168.610,44.581,158.340
C08278=1029.905,94.496,400.090,168.609,44.583,158.340
C08279=1029.899,94.246,400.109,168.606,44.585,158.340
C08280=1029.893,93.997,400.127,168.603,44.587,158.340
C08281=1029.887,93.748,400.147,168.601,44.589,158.340
C08282=1029.881,93.498,400.165,168.598,44.591,158.341
C08283=1029.875,93.249,400.185,168.596,44.593,158.341
C08284=1029.868,93.000,400.203,168.593,44.595,158.341
C08285=1029.862,92.751,400.222,168.591,44.597,158.341
C08286=1029.855,92.465,400.243,168.588,44.599,158.341
C08287=1029.849,92.180,400.265,168.586,44.602,158.342
C08288=1029.842,91.895,400.287,168.582,44.604,158.342
C08289=1029.835,91.610,400.308,168.580,44.607,158.342
C08290=1029.829,91.360,400.327,168.577,44.609,158.342
C08291=1029.823,91.112,400.345,168.575,44.610,158.342
C08292=1029.817,90.863,400.364,168.572,44.612,158.342
C08293=1029.811,90.614,400.383,168.571,44.615,158.343
C08294=1029.804,90.364,400.402,168.568,44.617,158.343
C08295=1029.799,90.115,400.421,168.566,44.619,158.343
C08296=1029.792,89.866,400.440,168.563,44.621,158.343
C08297=1029.787,89.616,400.459,168.561,44.623,158.343
C08298=1029.781,89.367,400.477,168.558,44.625,158.343
C08299=1029.774,89.118,400.496,168.556,44.627,158.344
C08300=1029.768,88.868,400.514,168.553,44.629,158.344
C08301=1029.761,88.619,400.533,168.550,44.631,158.344
C08302=1029.756,88.370,400.550,168.548,44.634,158.344
C08303=1029.749,88.121,400.569,168.546,44.636,158.344
C08304=1029.744,87.872,400.588,168.544,44.637,158.344
C08305=1029.737,87.623,400.607,168.542,44.640,158.345
C08306=1029.731,87.373,400.626,168.539,44.642,158.345
C08307=1029.725,87.124,400.643,168.537,44.644,158.345
C08308=1029.718,86.875,400.662,168.534,44.646,158.345
C08309=1029.712,86.625,400.681,168.532,44.648,158.345
C08310=1029.706,86.376,400.699,168.529,44.650,158.345
C08311=1029.700,86.127,400.717,168.526,44.652,158.346
C08312=1029.693,85.878,400.736,168.524,44.655,158.346
C08313=1029.688,85.629,400.755,168.522,44.657,158.346
C08314=1029.682,85.379,400.773,168.519,44.659,158.346
C08315=1029.675,85.130,400.791,168.518,44.661,158.346
C08316=1029.669,84.881,400.810,168.515,44.663,158.347
C08317=1029.663,84.632,400.828,168.513,44.665,158.347
C08318=1029.657,84.383,400.846,168.510,44.667,158.347
C08319=1029.650,84.133,400.865,168.508,44.670,158.347
C08320=1029.644,83.884,400.883,168.505,44.672,158.347
C08321=1029.638,83.635,400.902,168.502,44.674,158.347
C08322=1029.632,83.385,400.921,168.500,44.676,158.348
C08323=1029.627,83.136,400.938,168.498,44.678,158.348
C08324=1029.620,82.887,400.957,168.495,44.680,158.348
C08325=1029.614,82.637,400.975,168.493,44.682,158.348
C08326=1029.608,82.388,400.994,168.491,44.684,158.348
C08327=1029.601,82.139,401.012,168.489,44.686,158.349
C08328=1029.596,81.890,401.030,168.486,44.688,158.349
C08329=1029.589,81.641,401.048,168.483,44.690,158.349
C08330=1029.583,81.391,401.066,168.481,44.692,158.349
C08331=1029.577,81.142,401.085,168.478,44.694,158.349
C08332=1029.572,80.893,401.104,168.476,44.697,158.349
C08333=1029.566,80.644,401.122,168.473,44.699,158.349
C08334=1029.559,80.394,401.141,168.472,44.701,158.350
C08335=1029.553,80.145,401.158,168.469,44.703,158.350
C08336=1029.547,79.896,401.177,168.467,44.705,158.350
C08337=1029.541,79.647,401.195,168.464,44.707,158.350
C08338=1029.535,79.397,401.213,168.462,44.709,158.350
C08339=1029.529,79.148,401.231,168.459,44.711,158.350
C08340=1029.523,78.899,401.250,168.457,44.713,158.351
C08341=1029.517,78.649,401.267,168.455,44.715,158.351
C08342=1029.510,78.400,401.286,168.453,44.717,158.351
C08343=1029.505,78.150,401.305,168.450,44.719,158.351
C08344=1029.499,77.902,401.323,168.448,44.721,158.351
C08345=1029.493,77.652,401.341,168.445,44.723,158.351
C08346=1029.486,77.403,401.359,168.443,44.726,158.352
C08347=1029.480,77.154,401.377,168.440,44.728,158.352
C08348=1029.474,76.905,401.394,168.437,44.730,158.352
C08349=1029.468,76.655,401.413,168.435,44.732,158.352
C08350=1029.460,76.370,401.434,168.433,44.734,158.352
C08351=1029.453,76.085,401.454,168.430,44.737,158.353
C08352=1029.447,75.799,401.476,168.428,44.739,158.353
C08353=1029.440,75.514,401.495,168.424,44.742,158.353
C08354=1029.433,75.265,401.513,168.422,44.744,158.353
C08355=1029.427,75.015,401.531,168.419,44.746,158.353
C08356=1029.421,74.766,401.549,168.417,44.748,158.353
C08357=1029.415,74.517,401.567,168.415,44.750,158.354
C08358=1029.409,74.268,401.585,168.413,44.752,158.354
C08359=1029.403,74.018,401.603,168.410,44.755,158.354
C08360=1029.396,73.770,401.621,168.408,44.757,158.354
C08361=1029.390,73.520,401.639,168.405,44.758,158.354
C08362=1029.384,73.270,401.657,168.403,44.761,158.355
C08363=1029.378,73.021,401.674,168.400,44.763,158.355
C08364=1029.372,72.772,401.693,168.398,44.765,158.355
C08365=1029.365,72.523,401.710,168.395,44.767,158.355
C08366=1029.360,72.274,401.728,168.394,44.769,158.355
C08367=1029.353,72.024,401.747,168.391,44.771,158.355
C08368=1029.347,71.775,401.765,168.389,44.773,158.356
C08369=1029.342,71.526,401.782,168.386,44.775,158.356
C08370=1029.335,71.276,401.799,168.384,44.778,158.356
C08371=1029.329,71.027,401.817,168.381,44.780,158.356
C08372=1029.323,70.778,401.836,168.379,44.782,158.356
C08373=1029.317,70.528,401.854,168.376,44.784,158.356
C08374=1029.310,70.280,401.871,168.374,44.786,158.357
C08375=1029.304,70.030,401.889,168.372,44.788,158.357
C08376=1029.298,69.780,401.906,168.370,44.790,158.357
C08377=1029.293,69.531,401.924,168.367,44.793,158.357
C08378=1029.285,69.282,401.942,168.365,44.795,158.357
C08379=1029.280,69.033,401.960,168.362,44.797,158.357
C08380=1029.274,68.783,401.978,168.360,44.799,158.358
C08381=1029.268,68.534,401.996,168.357,44.801,158.358
C08382=1029.261,68.285,402.012,168.355,44.803,158.358
C08383=1029.255,68.035,402.030,168.352,44.805,158.358
C08384=1029.248,67.786,402.048,168.351,44.808,158.358
C08385=1029.243,67.537,402.065,168.348,44.810,158.358
C08386=1029.237,67.287,402.083,168.346,44.812,158.359
C08387=1029.231,67.038,402.100,168.343,44.814,158.359
C08388=1029.224,66.789,402.118,168.341,44.816,158.359
C08389=1029.219,66.540,402.136,168.338,44.818,158.359
C08390=1029.212,66.291,402.154,168.336,44.820,158.359
C08391=1029.206,66.041,402.172,168.333,44.823,158.360
C08392=1029.199,65.792,402.189,168.331,44.825,158.360
C08393=1029.193,65.543,402.207,168.328,44.827,158.360
C08394=1029.188,65.294,402.224,168.327,44.829,158.360
C08395=1029.181,65.044,402.242,168.324,44.831,158.360
C08396=1029.175,64.794,402.259,168.322,44.833,158.360
C08397=1029.168,64.546,402.276,168.319,44.835,158.360
C08398=1029.162,64.296,402.294,168.317,44.838,158.361
C08399=1029.156,64.047,402.311,168.314,44.840,158.361
C08400=1029.150,63.797,402.329,168.312,44.842,158.361
C08401=1029.144,63.548,402.346,168.309,44.844,158.361
C08402=1029.138,63.298,402.363,168.307,44.846,158.361
C08403=1029.132,63.050,402.380,168.304,44.848,158.361
C08404=1029.126,62.800,402.398,168.302,44.851,158.362
C08405=1029.119,62.550,402.416,168.299,44.853,158.362
C08406=1029.112,62.302,402.433,168.297,44.855,158.362
C08407=1029.106,62.052,402.449,168.295,44.857,158.362
C08408=1029.100,61.803,402.467,168.293,44.860,158.363
C08409=1029.093,61.553,402.484,168.291,44.862,158.363
C08410=1029.087,61.304,402.501,168.288,44.864,158.363
C08411=1029.080,61.055,402.519,168.286,44.866,158.363
C08412=1029.075,60.805,402.535,168.283,44.868,158.363
C08413=1029.068,60.556,402.553,168.281,44.871,158.364
C08414=1029.062,60.310,402.569,168.278,44.873,158.364
C08415=1029.056,60.063,402.587,168.276,44.876,158.364
C08416=1029.050,59.816,402.603,168.273,44.878,158.364
C08417=1029.043,59.569,402.620,168.271,44.879,158.364
C08418=1029.037,59.323,402.638,168.268,44.882,158.364
C08419=1029.031,59.076,402.655,168.266,44.884,158.365
C08420=1029.025,58.830,402.671,168.263,44.886,158.365
C08421=1029.019,58.584,402.689,168.262,44.889,158.365
C08422=1029.012,58.334,402.705,168.259,44.890,158.365
C08423=1029.006,58.085,402.722,168.257,44.893,158.365
C08424=1029.000,57.835,402.740,168.254,44.895,158.366
C08425=1028.994,57.587,402.757,168.252,44.897,158.366
C08426=1028.987,57.337,402.774,168.250,44.900,158.366
C08427=1028.981,57.088,402.791,168.247,44.902,158.366
C08428=1028.975,56.838,402.809,168.244,44.904,158.366
C08429=1028.969,56.589,402.825,168.242,44.906,158.366
C08430=1028.962,56.339,402.842,168.239,44.908,158.367
C08431=1028.956,56.091,402.859,168.237,44.910,158.367
C08432=1028.950,55.840,402.876,168.235,44.913,158.367
C08433=1028.944,55.591,402.893,168.232,44.915,158.367
C08434=1028.938,55.342,402.910,168.230,44.917,158.367
C08435=1028.931,55.093,402.927,168.227,44.919,158.367
C08436=1028.925,54.844,402.945,168.226,44.921,158.368
C08437=1028.919,54.594,402.961,168.223,44.924,158.368
C08438=1028.912,54.303,402.981,168.220,44.926,158.368
C08439=1028.904,54.012,403.001,168.217,44.929,158.368
C08440=1028.897,53.721,403.021,168.214,44.932,158.368
C08441=1028.889,53.430,403.041,168.211,44.934,158.369
C08442=1028.883,53.181,403.057,168.209,44.936,158.369
C08443=1028.878,52.932,403.075,168.207,44.938,158.369
C08444=1028.871,52.682,403.091,168.204,44.940,158.369
C08445=1028.865,52.433,403.108,168.202,44.943,158.369
C08446=1028.859,52.184,403.125,168.199,44.945,158.369
C08447=1028.853,51.934,403.142,168.198,44.947,158.370
C08448=1028.847,51.685,403.159,168.195,44.949,158.370
C08449=1028.840,51.435,403.176,168.193,44.951,158.370
C08450=1028.834,51.186,403.193,168.190,44.953,158.370
C08451=1028.829,50.937,403.210,168.188,44.955,158.370
C08452=1028.822,50.687,403.227,168.185,44.958,158.371
C08453=1028.816,50.438,403.243,168.183,44.960,158.371
C08454=1028.810,50.189,403.260,168.180,44.962,158.371
C08455=1028.803,49.939,403.277,168.177,44.964,158.371
C08456=1028.798,49.690,403.295,168.175,44.966,158.371
C08457=1028.792,49.441,403.311,168.173,44.968,158.371
C08458=1028.785,49.191,403.328,168.171,44.970,158.371
C08459=1028.779,48.942,403.344,168.169,44.973,158.372
C08460=1028.774,48.692,403.361,168.166,44.975,158.372
C08461=1028.767,48.443,403.379,168.164,44.977,158.372
C08462=1028.761,48.194,403.395,168.161,44.979,158.372
C08463=1028.755,47.945,403.412,168.158,44.981,158.372
C08464=1028.749,47.695,403.428,168.156,44.983,158.372
C08465=1028.742,47.446,403.446,168.154,44.985,158.373
C08466=1028.737,47.196,403.462,168.151,44.987,158.373
C08467=1028.731,46.947,403.479,168.149,44.989,158.373
C08468=1028.724,46.698,403.496,168.147,44.992,158.373
C08469=1028.718,46.448,403.513,168.145,44.994,158.373
C08470=1028.712,46.199,403.530,168.142,44.996,158.373
C08471=1028.706,45.950,403.546,168.139,44.998,158.373
C08472=1028.700,45.700,403.563,168.137,45.000,158.374
C08473=1028.693,45.451,403.580,168.135,45.002,158.374
C08474=1028.688,45.201,403.596,168.132,45.004,158.374
C08475=1028.682,44.952,403.613,168.129,45.006,158.374
C08476=1028.675,44.703,403.630,168.128,45.008,158.374
C08477=1028.669,44.453,403.646,168.125,45.010,158.374
C08478=1028.663,44.168,403.666,168.122,45.013,158.375
C08479=1028.656,43.882,403.685,168.119,45.015,158.375
C08480=1028.649,43.597,403.704,168.117,45.017,158.375
C08481=1028.642,43.310,403.723,168.113,45.020,158.375
C08482=1028.636,43.061,403.739,168.112,45.022,158.375
C08483=1028.630,42.812,403.757,168.110,45.024,158.375
C08484=1028.623,42.562,403.773,168.107,45.026,158.376
C08485=1028.617,42.313,403.789,168.104,45.028,158.376
C08486=1028.611,42.064,403.805,168.102,45.031,158.376
C08487=1028.605,41.814,403.821,168.100,45.033,158.376
C08488=1028.598,41.565,403.839,168.097,45.035,158.376
C08489=1028.593,41.315,403.855,168.095,45.037,158.376
C08490=1028.587,41.066,403.871,168.092,45.039,158.377
C08491=1028.581,40.817,403.888,168.090,45.041,158.377
C08492=1028.575,40.567,403.904,168.087,45.044,158.377
C08493=1028.568,40.317,403.920,168.085,45.046,158.377
C08494=1028.562,40.069,403.937,168.082,45.048,158.377
C08495=1028.556,39.819,403.954,168.080,45.050,158.377
C08496=1028.550,39.570,403.970,168.078,45.052,158.378
C08497=1028.544,39.321,403.986,168.076,45.054,158.378
C08498=1028.537,39.071,404.002,168.073,45.056,158.378
C08499=1028.531,38.821,404.018,168.071,45.059,158.378
C08500=1028.525,38.572,404.035,168.068,45.061,158.378
C08501=1028.519,38.323,404.051,168.066,45.063,158.378
C08502=1028.513,38.073,404.067,168.063,45.065,158.378
C08503=1028.507,37.824,404.083,168.061,45.068,158.379
C08504=1028.500,37.575,404.101,168.058,45.070,158.379
C08505=1028.494,37.325,404.117,168.056,45.072,158.379
C08506=1028.488,37.076,404.133,168.053,45.074,158.379
C08507=1028.482,36.827,404.150,168.051,45.076,158.379
C08508=1028.476,36.578,404.165,168.048,45.078,158.379
C08509=1028.470,36.328,404.181,168.046,45.081,158.380
C08510=1028.463,36.078,404.197,168.043,45.083,158.380
C08511=1028.457,35.828,404.213,168.041,45.085,158.380
C08512=1028.451,35.579,404.229,168.038,45.087,158.380
C08513=1028.445,35.330,404.246,168.036,45.089,158.380
C08514=1028.438,35.081,404.261,168.033,45.091,158.380
C08515=1028.432,34.831,404.277,168.031,45.094,158.381
C08516=1028.426,34.581,404.294,168.028,45.096,158.381
C08517=1028.420,34.332,404.310,168.026,45.099,158.381
C08518=1028.413,34.083,404.326,168.025,45.101,158.381
C08519=1028.407,33.834,404.342,168.022,45.103,158.381
C08520=1028.401,33.584,404.359,168.020,45.105,158.382
C08521=1028.395,33.335,404.373,168.017,45.107,158.382
C08522=1028.389,33.085,404.390,168.014,45.109,158.382
C08523=1028.383,32.836,404.406,168.012,45.112,158.382
C08524=1028.376,32.587,404.422,168.010,45.114,158.382
C08525=1028.370,32.337,404.438,168.007,45.116,158.382
C08526=1028.364,32.087,404.455,168.005,45.119,158.383
C08527=1028.357,31.838,404.470,168.002,45.121,158.383
C08528=1028.351,31.588,404.486,168.000,45.122,158.383
C08529=1028.345,31.339,404.502,167.997,45.125,158.383
C08530=1028.339,31.090,404.518,167.995,45.127,158.383
C08531=1028.333,30.841,404.534,167.992,45.129,158.383
C08532=1028.327,30.591,404.550,167.990,45.132,158.384
C08533=1028.320,30.342,404.565,167.987,45.134,158.384
C08534=1028.314,30.092,404.581,167.985,45.136,158.384
C08535=1028.308,29.843,404.598,167.982,45.138,158.384
C08536=1028.302,29.594,404.613,167.980,45.140,158.384
C08537=1028.296,29.345,404.630,167.977,45.142,158.384
C08538=1028.290,29.095,404.645,167.975,45.144,158.384
C08539=1028.283,28.846,404.661,167.972,45.147,158.385
C08540=1028.277,28.596,404.677,167.970,45.149,158.385
C08541=1028.272,28.346,404.693,167.967,45.151,158.385
C08542=1028.264,28.060,404.711,167.965,45.154,158.385
C08543=1028.257,27.775,404.729,167.961,45.156,158.385
C08544=1028.250,27.489,404.747,167.959,45.159,158.385
C08545=1028.243,27.203,404.766,167.957,45.161,158.386
C08546=1028.236,26.953,404.781,167.954,45.163,158.386
C08547=1028.230,26.704,404.797,167.952,45.166,158.386
C08548=1028.224,26.455,404.813,167.949,45.168,158.386
C08549=1028.217,26.205,404.828,167.947,45.170,158.386
C08550=1028.211,25.956,404.844,167.944,45.173,158.387
C08551=1028.205,25.706,404.859,167.942,45.175,158.387
C08552=1028.199,25.457,404.875,167.939,45.177,158.387
C08553=1028.192,25.208,404.891,167.937,45.179,158.387
C08554=1028.187,24.958,404.906,167.934,45.181,158.387
C08555=1028.180,24.709,404.922,167.932,45.183,158.387
C08556=1028.174,24.459,404.937,167.930,45.186,158.388
C08557=1028.168,24.210,404.953,167.927,45.188,158.388
C08558=1028.161,23.960,404.968,167.925,45.191,158.388
C08559=1028.155,23.711,404.984,167.922,45.193,158.388
C08560=1028.150,23.462,404.999,167.920,45.195,158.388
C08561=1028.144,23.213,405.015,167.917,45.197,158.388
C08562=1028.137,22.963,405.030,167.915,45.199,158.388
C08563=1028.131,22.714,405.046,167.912,45.201,158.389
C08564=1028.125,22.464,405.061,167.910,45.204,158.389
C08565=1028.118,22.215,405.077,167.907,45.206,158.389
C08566=1028.113,21.965,405.092,167.905,45.208,158.389
C08567=1028.106,21.716,405.108,167.902,45.211,158.389
C08568=1028.100,21.466,405.124,167.900,45.213,158.389
C08569=1028.094,21.217,405.139,167.897,45.215,158.390
C08570=1028.087,20.967,405.154,167.895,45.217,158.390
C08571=1028.081,20.718,405.171,167.892,45.219,158.390
C08572=1028.075,20.468,405.186,167.890,45.221,158.390
C08573=1028.069,20.219,405.202,167.887,45.223,158.390
C08574=1028.062,19.969,405.217,167.885,45.226,158.390
C08575=1028.057,19.720,405.231,167.882,45.228,158.391
C08576=1028.051,19.471,405.248,167.879,45.230,158.391
C08577=1028.044,19.221,405.262,167.876,45.233,158.391
C08578=1028.038,18.972,405.278,167.874,45.235,158.391
C08579=1028.032,18.722,405.294,167.872,45.238,158.391
C08580=1028.026,18.473,405.309,167.869,45.240,158.391
C08581=1028.019,18.224,405.324,167.866,45.242,158.391
C08582=1028.013,17.974,405.339,167.864,45.244,158.392
C08583=1028.007,17.724,405.355,167.862,45.246,158.392
C08584=1028.001,17.476,405.370,167.859,45.248,158.392
C08585=1027.994,17.226,405.385,167.857,45.251,158.392
C08586=1027.989,16.976,405.401,167.854,45.253,158.392
C08587=1027.982,16.726,405.416,167.852,45.255,158.392
C08588=1027.976,16.477,405.431,167.849,45.258,158.393
C08589=1027.969,16.228,405.446,167.847,45.260,158.393
C08590=1027.964,15.978,405.462,167.844,45.262,158.393
C08591=1027.958,15.729,405.477,167.842,45.264,158.393
C08592=1027.951,15.480,405.492,167.839,45.266,158.393
C08593=1027.945,15.230,405.507,167.837,45.268,158.393
C08594=1027.939,14.980,405.522,167.834,45.271,158.394
C08595=1027.933,14.731,405.538,167.832,45.273,158.394
C08596=1027.926,14.481,405.553,167.829,45.275,158.394
C08597=1027.920,14.232,405.568,167.827,45.278,158.394
C08598=1027.915,13.983,405.583,167.824,45.280,158.394
C08599=1027.908,13.733,405.598,167.822,45.282,158.394
C08600=1027.902,13.483,405.613,167.819,45.284,158.394
C08601=1027.895,13.234,405.629,167.817,45.286,158.395
C08602=1027.889,12.984,405.644,167.815,45.289,158.395
C08603=1027.883,12.736,405.658,167.811,45.291,158.395
C08604=1027.877,12.486,405.673,167.809,45.294,158.395
C08605=1027.870,12.236,405.688,167.806,45.296,158.395
C08606=1027.863,11.952,405.705,167.804,45.299,158.396
C08607=1027.856,11.668,405.722,167.800,45.302,158.396
C08608=1027.849,11.383,405.739,167.798,45.304,158.396
C08609=1027.841,11.098,405.755,167.795,45.307,158.396
C08610=1027.835,10.849,405.770,167.792,45.309,158.396
C08611=1027.829,10.599,405.785,167.790,45.311,158.396
C08612=1027.823,10.350,405.800,167.787,45.313,158.396
C08613=1027.816,10.101,405.816,167.785,45.316,158.397
C08614=1027.810,9.851,405.831,167.782,45.318,158.397
C08615=1027.803,9.602,405.845,167.780,45.321,158.397
C08616=1027.798,9.353,405.860,167.776,45.323,158.397
C08617=1027.791,9.103,405.875,167.774,45.326,158.397
C08618=1027.785,8.853,405.889,167.772,45.328,158.398
C08619=1027.779,8.603,405.904,167.769,45.330,158.398
C08620=1027.773,8.354,405.919,167.767,45.332,158.398
C08621=1027.767,8.104,405.934,167.764,45.334,158.398
C08622=1027.760,7.855,405.949,167.762,45.337,158.398
C08623=1027.754,7.605,405.964,167.759,45.339,158.398
C08624=1027.748,7.356,405.978,167.757,45.341,158.398
C08625=1027.742,7.107,405.993,167.754,45.344,158.399
C08626=1027.735,6.857,406.008,167.752,45.346,158.399
C08627=1027.729,6.607,406.023,167.748,45.349,158.399
C08628=1027.723,6.358,406.038,167.746,45.351,158.399
C08629=1027.717,6.109,406.053,167.743,45.353,158.399
C08630=1027.710,5.859,406.067,167.741,45.355,158.399
C08631=1027.705,5.610,406.082,167.738,45.357,158.400
C08632=1027.698,5.360,406.096,167.736,45.359,158.400
C08633=1027.691,5.110,406.111,167.734,45.362,158.400
C08634=1027.686,4.861,406.125,167.731,45.364,158.400
C08635=1027.679,4.612,406.140,167.728,45.366,158.400
C08636=1027.673,4.362,406.155,167.726,45.369,158.400
C08637=1027.667,4.113,406.170,167.724,45.371,158.400
C08638=1027.661,3.863,406.185,167.721,45.373,158.401
C08639=1027.655,3.613,406.199,167.718,45.376,158.401
C08640=1027.649,3.364,406.213,167.715,45.378,158.401
C08641=1027.642,3.115,406.228,167.713,45.380,158.401
C08642=1027.637,2.866,406.243,167.710,45.382,158.401
C08643=1027.630,2.616,406.258,167.708,45.384,158.401
C08644=1027.624,2.366,406.272,167.705,45.386,158.401
C08645=1027.618,2.117,406.287,167.703,45.389,158.402
C08646=1027.612,1.867,406.302,167.700,45.391,158.402
C08647=1027.606,1.617,406.317,167.698,45.393,158.402
C08648=1027.600,1.368,406.331,167.695,45.396,158.402
C08649=1027.593,1.119,406.345,167.693,45.398,158.402
C08650=1027.587,0.870,406.359,167.690,45.400,158.402
C08651=1027.581,0.620,406.374,167.687,45.403,158.403
C08652=1027.574,0.370,406.389,167.684,45.405,158.403
C08653=1027.569,0.121,406.403,167.682,45.407,158.403
C08654=1027.563,-0.129,406.418,167.679,45.409,158.403
C08655=1027.557,-0.378,406.433,167.677,45.412,158.403
C08656=1027.551,-0.628,406.447,167.674,45.414,158.403
C08657=1027.545,-0.877,406.462,167.672,45.416,158.403
C08658=1027.539,-1.127,406.476,167.669,45.418,158.403
C08659=1027.533,-1.376,406.491,167.667,45.420,158.404
C08660=1027.527,-1.626,406.505,167.664,45.422,158.404
C08661=1027.521,-1.875,406.520,167.662,45.424,158.404
C08662=1027.514,-2.124,406.534,167.660,45.427,158.404
C08663=1027.508,-2.375,406.548,167.656,45.429,158.404
C08664=1027.502,-2.624,406.563,167.653,45.431,158.404
C08665=1027.496,-2.874,406.577,167.651,45.433,158.404
C08666=1027.490,-3.123,406.592,167.648,45.435,158.404
C08667=1027.484,-3.372,406.607,167.646,45.438,158.405
C08668=1027.478,-3.622,406.621,167.643,45.440,158.405
C08669=1027.472,-3.872,406.636,167.641,45.442,158.405
C08670=1027.465,-4.154,406.651,167.638,45.445,158.405
C08671=1027.458,-4.436,406.668,167.635,45.448,158.405
C08672=1027.451,-4.719,406.683,167.632,45.450,158.405
C08673=1027.444,-5.002,406.699,167.629,45.453,158.406
C08674=1027.437,-5.251,406.713,167.626,45.456,158.406
C08675=1027.432,-5.500,406.727,167.624,45.458,158.406
C08676=1027.425,-5.750,406.742,167.621,45.460,158.406
C08677=1027.419,-5.999,406.755,167.619,45.462,158.406
C08678=1027.413,-6.249,406.770,167.616,45.464,158.406
C08679=1027.406,-6.498,406.784,167.614,45.467,158.407
C08680=1027.400,-6.749,406.798,167.610,45.469,158.407
C08681=1027.394,-6.997,406.812,167.608,45.472,158.407
C08682=1027.388,-7.247,406.826,167.605,45.474,158.407
C08683=1027.382,-7.496,406.841,167.603,45.477,158.407
C08684=1027.375,-7.746,406.854,167.600,45.479,158.407
C08685=1027.370,-7.996,406.868,167.598,45.481,158.407
C08686=1027.363,-8.245,406.883,167.595,45.484,158.408
C08687=1027.357,-8.495,406.896,167.592,45.486,158.408
C08688=1027.350,-8.744,406.911,167.590,45.488,158.408
C08689=1027.344,-8.994,406.925,167.587,45.490,158.408
C08690=1027.338,-9.244,406.938,167.585,45.492,158.408
C08691=1027.332,-9.493,406.953,167.581,45.495,158.408
C08692=1027.326,-9.742,406.967,167.579,45.497,158.408
C08693=1027.320,-9.992,406.980,167.576,45.500,158.409
C08694=1027.314,-10.241,406.995,167.574,45.502,158.409
C08695=1027.307,-10.491,407.009,167.571,45.504,158.409
C08696=1027.301,-10.741,407.022,167.569,45.507,158.409
C08697=1027.295,-10.991,407.036,167.565,45.509,158.409
C08698=1027.289,-11.240,407.051,167.563,45.511,158.409
C08699=1027.283,-11.489,407.064,167.561,45.514,158.410
C08700=1027.277,-11.739,407.078,167.558,45.516,158.410
C08701=1027.270,-11.988,407.092,167.555,45.518,158.410
C08702=1027.265,-12.237,407.106,167.553,45.521,158.410
C08703=1027.259,-12.488,407.120,167.550,45.523,158.410
C08704=1027.252,-12.737,407.134,167.547,45.526,158.410
C08705=1027.246,-12.987,407.148,167.545,45.528,158.410
C08706=1027.240,-13.236,407.162,167.542,45.530,158.410
C08707=1027.234,-13.485,407.176,167.540,45.532,158.411
C08708=1027.227,-13.735,407.189,167.537,45.534,158.411
C08709=1027.222,-13.985,407.203,167.534,45.537,158.411
C08710=1027.215,-14.234,407.217,167.531,45.539,158.411
C08711=1027.209,-14.484,407.231,167.529,45.541,158.411
C08712=1027.203,-14.733,407.245,167.526,45.543,158.411
C08713=1027.198,-14.983,407.258,167.524,45.545,158.411
C08714=1027.191,-15.233,407.272,167.521,45.548,158.412
C08715=1027.185,-15.482,407.286,167.518,45.550,158.412
C08716=1027.179,-15.732,407.299,167.515,45.552,158.412
C08717=1027.173,-15.982,407.313,167.513,45.555,158.412
C08718=1027.167,-16.231,407.327,167.510,45.557,158.412
C08719=1027.160,-16.480,407.341,167.507,45.560,158.412
C08720=1027.154,-16.730,407.354,167.505,45.562,158.412
C08721=1027.148,-16.979,407.368,167.502,45.565,158.413
C08722=1027.142,-17.229,407.381,167.500,45.567,158.413
C08723=1027.135,-17.479,407.395,167.496,45.570,158.413
C08724=1027.130,-17.728,407.409,167.494,45.572,158.413
C08725=1027.123,-17.977,407.422,167.492,45.574,158.413
C08726=1027.117,-18.227,407.436,167.489,45.577,158.413
C08727=1027.110,-18.477,407.449,167.487,45.579,158.414
C08728=1027.105,-18.726,407.463,167.483,45.581,158.414
C08729=1027.099,-18.975,407.476,167.481,45.584,158.414
C08730=1027.092,-19.226,407.489,167.478,45.586,158.414
C08731=1027.086,-19.475,407.502,167.476,45.588,158.414
C08732=1027.080,-19.725,407.516,167.472,45.591,158.414
C08733=1027.074,-19.974,407.530,167.470,45.593,158.414
C08734=1027.067,-20.255,407.545,167.466,45.596,158.414
C08735=1027.060,-20.536,407.560,167.464,45.599,158.415
C08736=1027.054,-20.817,407.575,167.461,45.601,158.415
C08737=1027.046,-21.098,407.590,167.457,45.604,158.415
C08738=1027.040,-21.347,407.604,167.455,45.607,158.415
C08739=1027.034,-21.597,407.617,167.452,45.609,158.415
C08740=1027.027,-21.847,407.631,167.450,45.611,158.415
C08741=1027.021,-22.096,407.644,167.448,45.614,158.416
C08742=1027.015,-22.346,407.657,167.444,45.616,158.416
C08743=1027.010,-22.595,407.671,167.442,45.619,158.416
C08744=1027.004,-22.845,407.684,167.439,45.621,158.416
C08745=1026.997,-23.095,407.698,167.437,45.623,158.416
C08746=1026.991,-23.344,407.711,167.433,45.626,158.416
C08747=1026.985,-23.593,407.725,167.431,45.628,158.416
C08748=1026.979,-23.843,407.737,167.428,45.630,158.416
C08749=1026.973,-24.093,407.751,167.426,45.632,158.417
C08750=1026.967,-24.342,407.764,167.422,45.635,158.417
C08751=1026.961,-24.592,407.778,167.420,45.637,158.417
C08752=1026.954,-24.841,407.791,167.417,45.639,158.417
C08753=1026.949,-25.091,407.804,167.415,45.641,158.417
C08754=1026.942,-25.341,407.817,167.412,45.644,158.417
C08755=1026.936,-25.590,407.830,167.409,45.646,158.417
C08756=1026.931,-25.839,407.844,167.406,45.648,158.418
C08757=1026.924,-26.089,407.858,167.404,45.651,158.418
C08758=1026.918,-26.339,407.871,167.401,45.653,158.418
C08759=1026.912,-26.589,407.884,167.398,45.655,158.418
C08760=1026.906,-26.838,407.898,167.396,45.658,158.418
C08761=1026.900,-27.088,407.910,167.393,45.660,158.418
C08762=1026.894,-27.337,407.923,167.390,45.662,158.418
C08763=1026.888,-27.586,407.937,167.387,45.665,158.418
C08764=1026.882,-27.836,407.949,167.385,45.667,158.419
C08765=1026.876,-28.086,407.963,167.381,45.670,158.419
C08766=1026.870,-28.335,407.976,167.379,45.672,158.419
C08767=1026.863,-28.586,407.989,167.377,45.675,158.419
C08768=1026.857,-28.835,408.002,167.374,45.677,158.419
C08769=1026.851,-29.085,408.015,167.371,45.680,158.419
C08770=1026.845,-29.334,408.028,167.368,45.682,158.419
C08771=1026.839,-29.584,408.040,167.366,45.685,158.420
C08772=1026.833,-29.833,408.054,167.362,45.687,158.420
C08773=1026.827,-30.083,408.066,167.360,45.690,158.420
C08774=1026.820,-30.332,408.079,167.357,45.692,158.420
C08775=1026.814,-30.581,408.093,167.354,45.695,158.420
C08776=1026.808,-30.831,408.105,167.351,45.697,158.420
C08777=1026.801,-31.080,408.118,167.349,45.699,158.421
C08778=1026.795,-31.330,408.131,167.346,45.702,158.421
C08779=1026.789,-31.579,408.144,167.343,45.704,158.421
C08780=1026.783,-31.830,408.157,167.341,45.707,158.421
C08781=1026.777,-32.079,408.170,167.337,45.709,158.421
C08782=1026.771,-32.329,408.183,167.335,45.712,158.421
C08783=1026.765,-32.579,408.195,167.333,45.714,158.421
C08784=1026.759,-32.828,408.208,167.330,45.716,158.421
C08785=1026.753,-33.078,408.221,167.327,45.719,158.422
C08786=1026.746,-33.327,408.234,167.324,45.721,158.422
C08787=1026.741,-33.577,408.247,167.322,45.723,158.422
C08788=1026.734,-33.827,408.260,167.318,45.726,158.422
C08789=1026.728,-34.077,408.273,167.316,45.728,158.422
C08790=1026.722,-34.326,408.285,167.313,45.731,158.422
C08791=1026.716,-34.576,408.298,167.310,45.733,158.422
C08792=1026.710,-34.826,408.311,167.308,45.736,158.423
C08793=1026.703,-35.074,408.324,167.305,45.738,158.423
C08794=1026.697,-35.324,408.336,167.301,45.740,158.423
C08795=1026.692,-35.574,408.348,167.299,45.743,158.423
C08796=1026.686,-35.823,408.362,167.297,45.745,158.423
C08797=1026.680,-36.073,408.374,167.293,45.748,158.423
C08798=1026.673,-36.353,408.389,167.291,45.750,158.423
C08799=1026.666,-36.633,408.403,167.287,45.753,158.423
C08800=1026.660,-36.913,408.417,167.284,45.756,158.424
C08801=1026.653,-37.194,408.432,167.282,45.759,158.424
C08802=1026.647,-37.443,408.445,167.278,45.761,158.424
C08803=1026.641,-37.693,408.457,167.276,45.763,158.424
C08804=1026.635,-37.942,408.469,167.273,45.766,158.424
C08805=1026.629,-38.191,408.482,167.270,45.768,158.424
C08806=1026.623,-38.441,408.495,167.267,45.771,158.424
C08807=1026.617,-38.691,408.507,167.265,45.773,158.425
C08808=1026.611,-38.940,408.520,167.261,45.775,158.425
C08809=1026.605,-39.190,408.533,167.259,45.778,158.425
C08810=1026.599,-39.440,408.546,167.257,45.780,158.425
C08811=1026.592,-39.689,408.558,167.253,45.783,158.425
C08812=1026.586,-39.939,408.570,167.251,45.785,158.425
C08813=1026.580,-40.189,408.583,167.247,45.788,158.425
C08814=1026.574,-40.439,408.595,167.245,45.791,158.426
C08815=1026.568,-40.688,408.607,167.242,45.793,158.426
C08816=1026.562,-40.937,408.620,167.239,45.796,158.426
C08817=1026.555,-41.187,408.632,167.237,45.798,158.426
C08818=1026.550,-41.436,408.645,167.233,45.801,158.426
C08819=1026.544,-41.686,408.657,167.231,45.803,158.426
C08820=1026.537,-41.936,408.669,167.228,45.806,158.426
C08821=1026.531,-42.186,408.682,167.225,45.808,158.426
C08822=1026.525,-42.435,408.693,167.223,45.811,158.427
C08823=1026.519,-42.685,408.706,167.220,45.813,158.427
C08824=1026.513,-42.934,408.718,167.217,45.816,158.427
C08825=1026.507,-43.184,408.730,167.214,45.818,158.427
C08826=1026.501,-43.434,408.743,167.211,45.821,158.427
C08827=1026.495,-43.684,408.756,167.208,45.823,158.427
C08828=1026.489,-43.933,408.767,167.206,45.825,158.428
C08829=1026.483,-44.183,408.780,167.202,45.828,158.428
C08830=1026.477,-44.432,408.792,167.200,45.830,158.428
C08831=1026.470,-44.682,408.804,167.197,45.833,158.428
C08832=1026.464,-44.932,408.817,167.194,45.835,158.428
C08833=1026.458,-45.181,408.828,167.192,45.837,158.428
C08834=1026.452,-45.431,408.841,167.188,45.840,158.428
C08835=1026.447,-45.680,408.853,167.186,45.842,158.428
C08836=1026.440,-45.930,408.865,167.183,45.845,158.429
C08837=1026.435,-46.179,408.878,167.180,45.847,158.429
C08838=1026.429,-46.429,408.890,167.178,45.850,158.429
C08839=1026.422,-46.679,408.902,167.174,45.853,158.429
C08840=1026.416,-46.929,408.915,167.172,45.855,158.429
C08841=1026.410,-47.177,408.926,167.169,45.857,158.429
C08842=1026.404,-47.427,408.939,167.166,45.860,158.429
C08843=1026.398,-47.677,408.951,167.163,45.862,158.429
C08844=1026.392,-47.927,408.963,167.160,45.865,158.430
C08845=1026.386,-48.176,408.975,167.158,45.867,158.430
C08846=1026.381,-48.426,408.987,167.155,45.870,158.430
C08847=1026.374,-48.676,408.999,167.152,45.872,158.430
C08848=1026.369,-48.925,409.011,167.149,45.874,158.430
C08849=1026.362,-49.175,409.023,167.146,45.877,158.430
C08850=1026.356,-49.425,409.036,167.143,45.879,158.430
C08851=1026.351,-49.674,409.048,167.141,45.882,158.431
C08852=1026.344,-49.923,409.060,167.137,45.885,158.431
C08853=1026.339,-50.174,409.072,167.135,45.887,158.431
C08854=1026.332,-50.424,409.084,167.133,45.889,158.431
C08855=1026.327,-50.673,409.096,167.129,45.892,158.431
C08856=1026.320,-50.922,409.108,167.127,45.894,158.431
C08857=1026.314,-51.173,409.120,167.123,45.897,158.431
C08858=1026.308,-51.422,409.132,167.121,45.900,158.431
C08859=1026.302,-51.671,409.143,167.117,45.902,158.431
C08860=1026.295,-51.921,409.155,167.115,45.905,158.432
C08861=1026.290,-52.171,409.167,167.112,45.908,158.432
C08862=1026.283,-52.452,409.180,167.109,45.911,158.432
C08863=1026.275,-52.732,409.193,167.105,45.914,158.432
C08864=1026.269,-53.012,409.206,167.102,45.917,158.432
C08865=1026.262,-53.293,409.220,167.099,45.920,158.433
C08866=1026.256,-53.542,409.231,167.096,45.922,158.433
C08867=1026.250,-53.792,409.242,167.093,45.925,158.433
C08868=1026.243,-54.042,409.254,167.090,45.928,158.433
C08869=1026.238,-54.291,409.266,167.087,45.930,158.433
C08870=1026.231,-54.541,409.278,167.085,45.933,158.433
C08871=1026.225,-54.791,409.289,167.081,45.936,158.433
C08872=1026.219,-55.040,409.301,167.079,45.938,158.433
C08873=1026.212,-55.290,409.313,167.075,45.941,158.434
C08874=1026.207,-55.539,409.324,167.073,45.944,158.434
C08875=1026.201,-55.789,409.336,167.070,45.946,158.434
C08876=1026.194,-56.039,409.347,167.067,45.949,158.434
C08877=1026.188,-56.288,409.359,167.064,45.952,158.434
C08878=1026.182,-56.538,409.370,167.061,45.954,158.434
C08879=1026.177,-56.787,409.382,167.058,45.957,158.435
C08880=1026.170,-57.038,409.394,167.056,45.959,158.435
C08881=1026.164,-57.287,409.405,167.052,45.962,158.435
C08882=1026.158,-57.537,409.416,167.050,45.965,158.435
C08883=1026.152,-57.787,409.428,167.047,45.967,158.435
C08884=1026.146,-58.036,409.440,167.044,45.970,158.435
C08885=1026.140,-58.286,409.451,167.041,45.973,158.435
C08886=1026.134,-58.535,409.463,167.038,45.975,158.436
C08887=1026.128,-58.785,409.474,167.035,45.978,158.436
C08888=1026.122,-59.034,409.485,167.033,45.980,158.436
C08889=1026.116,-59.285,409.497,167.029,45.983,158.436
C08890=1026.110,-59.534,409.508,167.027,45.985,158.436
C08891=1026.104,-59.784,409.520,167.023,45.988,158.436
C08892=1026.098,-60.033,409.531,167.021,45.990,158.436
C08893=1026.091,-60.283,409.543,167.018,45.993,158.437
C08894=1026.086,-60.533,409.554,167.015,45.996,158.437
C08895=1026.080,-60.783,409.566,167.012,45.999,158.437
C08896=1026.074,-61.032,409.577,167.009,46.001,158.437
C08897=1026.067,-61.282,409.589,167.007,46.003,158.437
C08898=1026.062,-61.531,409.599,167.004,46.006,158.437
C08899=1026.056,-61.781,409.612,167.001,46.009,158.437
C08900=1026.050,-62.031,409.623,166.998,46.011,158.437
C08901=1026.044,-62.280,409.634,166.995,46.014,158.438
C08902=1026.038,-62.530,409.645,166.992,46.016,158.438
C08903=1026.032,-62.779,409.657,166.990,46.019,158.438
C08904=1026.026,-63.029,409.668,166.986,46.022,158.438
C08905=1026.021,-63.279,409.679,166.984,46.024,158.438
C08906=1026.014,-63.529,409.691,166.980,46.027,158.438
C08907=1026.008,-63.778,409.702,166.978,46.029,158.438
C08908=1026.002,-64.028,409.713,166.975,46.032,158.439
C08909=1025.996,-64.278,409.724,166.972,46.034,158.439
C08910=1025.990,-64.527,409.736,166.969,46.037,158.439
C08911=1025.984,-64.777,409.748,166.966,46.040,158.439
C08912=1025.979,-65.027,409.759,166.963,46.042,158.439
C08913=1025.973,-65.276,409.769,166.961,46.045,158.439
C08914=1025.967,-65.527,409.781,166.957,46.048,158.439
C08915=1025.961,-65.775,409.792,166.955,46.050,158.439
C08916=1025.955,-66.025,409.803,166.951,46.053,158.439
C08917=1025.948,-66.275,409.814,166.949,46.055,158.440
C08918=1025.943,-66.525,409.826,166.946,46.058,158.440
C08919=1025.938,-66.774,409.837,166.943,46.060,158.440
C08920=1025.931,-67.025,409.848,166.940,46.063,158.440
C08921=1025.925,-67.273,409.860,166.937,46.065,158.440
C08922=1025.920,-67.523,409.870,166.934,46.068,158.440
C08923=1025.913,-67.773,409.882,166.931,46.071,158.440
C08924=1025.908,-68.023,409.893,166.928,46.074,158.441
C08925=1025.903,-68.272,409.904,166.925,46.076,158.441
C08926=1025.896,-68.554,409.916,166.922,46.079,158.441
C08927=1025.889,-68.835,409.929,166.919,46.082,158.441
C08928=1025.882,-69.117,409.941,166.915,46.085,158.441
C08929=1025.876,-69.399,409.954,166.912,46.088,158.441
C08930=1025.870,-69.649,409.965,166.909,46.090,158.441
C08931=1025.864,-69.899,409.976,166.906,46.093,158.441
C08932=1025.858,-70.148,409.987,166.903,46.095,158.441
C08933=1025.852,-70.397,409.999,166.900,46.098,158.442
C08934=1025.846,-70.647,410.010,166.897,46.100,158.442
C08935=1025.840,-70.897,410.021,166.895,46.103,158.442
C08936=1025.835,-71.147,410.032,166.891,46.106,158.442
C08937=1025.830,-71.396,410.043,166.889,46.108,158.442
C08938=1025.823,-71.646,410.054,166.885,46.111,158.442
C08939=1025.817,-71.896,410.065,166.883,46.113,158.442
C08940=1025.812,-72.145,410.076,166.880,46.116,158.443
C08941=1025.806,-72.395,410.087,166.877,46.118,158.443
C08942=1025.800,-72.644,410.098,166.874,46.121,158.443
C08943=1025.794,-72.895,410.108,166.871,46.123,158.443
C08944=1025.788,-73.145,410.119,166.868,46.126,158.443
C08945=1025.783,-73.394,410.131,166.865,46.128,158.443
C08946=1025.778,-73.644,410.142,166.862,46.131,158.443
C08947=1025.771,-73.894,410.153,166.859,46.133,158.443
C08948=1025.766,-74.143,410.164,166.856,46.136,158.443
C08949=1025.760,-74.393,410.175,166.854,46.138,158.444
C08950=1025.754,-74.642,410.186,166.850,46.141,158.444
C08951=1025.749,-74.893,410.196,166.848,46.144,158.444
C08952=1025.742,-75.142,410.206,166.844,46.146,158.444
C08953=1025.736,-75.392,410.217,166.842,46.149,158.444
C08954=1025.730,-75.641,410.228,166.839,46.152,158.444
C08955=1025.724,-75.891,410.239,166.835,46.155,158.444
C08956=1025.719,-76.141,410.249,166.833,46.157,158.445
C08957=1025.713,-76.391,410.260,166.830,46.160,158.445
C08958=1025.706,-76.640,410.271,166.827,46.162,158.445
C08959=1025.700,-76.890,410.282,166.824,46.165,158.445
C08960=1025.695,-77.140,410.292,166.822,46.168,158.445
C08961=1025.689,-77.390,410.303,166.818,46.171,158.445
C08962=1025.684,-77.639,410.313,166.815,46.174,158.445
C08963=1025.677,-77.889,410.323,166.812,46.176,158.445
C08964=1025.672,-78.138,410.334,166.809,46.179,158.445
C08965=1025.666,-78.388,410.345,166.807,46.181,158.446
C08966=1025.660,-78.638,410.355,166.803,46.184,158.446
C08967=1025.654,-78.888,410.366,166.801,46.187,158.446
C08968=1025.648,-79.137,410.376,166.797,46.190,158.446
C08969=1025.642,-79.387,410.387,166.794,46.193,158.446
C08970=1025.636,-79.637,410.398,166.792,46.195,158.446
C08971=1025.631,-79.886,410.408,166.788,46.198,158.446
C08972=1025.625,-80.136,410.419,166.786,46.200,158.447
C08973=1025.619,-80.386,410.429,166.783,46.203,158.447
C08974=1025.613,-80.636,410.439,166.779,46.206,158.447
C08975=1025.607,-80.885,410.449,166.777,46.209,158.447
C08976=1025.601,-81.135,410.459,166.773,46.212,158.447
C08977=1025.594,-81.385,410.470,166.770,46.215,158.447
C08978=1025.589,-81.635,410.480,166.768,46.217,158.448
C08979=1025.583,-81.885,410.491,166.765,46.220,158.448
C08980=1025.577,-82.134,410.501,166.762,46.222,158.448
C08981=1025.571,-82.384,410.512,166.759,46.225,158.448
C08982=1025.565,-82.634,410.521,166.755,46.228,158.448
C08983=1025.559,-82.883,410.532,166.753,46.231,158.448
C08984=1025.553,-83.133,410.542,166.750,46.234,158.448
C08985=1025.547,-83.382,410.552,166.747,46.237,158.449
C08986=1025.541,-83.632,410.562,166.744,46.239,158.449
C08987=1025.536,-83.882,410.572,166.741,46.242,158.449
C08988=1025.529,-84.131,410.582,166.737,46.245,158.449
C08989=1025.524,-84.382,410.593,166.735,46.248,158.449
C08990=1025.517,-84.665,410.604,166.732,46.251,158.449
C08991=1025.511,-84.948,410.616,166.727,46.254,158.449
C08992=1025.503,-85.233,410.627,166.724,46.258,158.450
C08993=1025.497,-85.517,410.639,166.721,46.261,158.450
C08994=1025.491,-85.767,410.648,166.719,46.263,158.450
C08995=1025.485,-86.016,410.659,166.715,46.266,158.450
C08996=1025.480,-86.266,410.669,166.712,46.269,158.450
C08997=1025.474,-86.516,410.679,166.710,46.272,158.450
C08998=1025.468,-86.765,410.690,166.706,46.275,158.451
C08999=1025.462,-87.015,410.699,166.703,46.277,158.451
C09000=1025.456,-87.265,410.710,166.701,46.280,158.451
C09001=1025.450,-87.514,410.719,166.697,46.283,158.451
C09002=1025.445,-87.764,410.730,166.694,46.286,158.451
C09003=1025.439,-88.014,410.739,166.691,46.288,158.451
C09004=1025.433,-88.263,410.750,166.688,46.291,158.451
C09005=1025.427,-88.513,410.760,166.685,46.294,158.451
C09006=1025.421,-88.763,410.770,166.683,46.297,158.452
C09007=1025.415,-89.013,410.779,166.679,46.300,158.452
C09008=1025.409,-89.262,410.790,166.677,46.302,158.452
C09009=1025.403,-89.512,410.800,166.673,46.305,158.452
C09010=1025.398,-89.762,410.810,166.670,46.308,158.452
C09011=1025.392,-90.011,410.819,166.668,46.311,158.452
C09012=1025.387,-90.262,410.829,166.664,46.314,158.452
C09013=1025.380,-90.511,410.840,166.661,46.317,158.452
C09014=1025.375,-90.761,410.850,166.659,46.319,158.453
C09015=1025.369,-91.011,410.859,166.655,46.322,158.453
C09016=1025.363,-91.261,410.870,166.652,46.325,158.453
C09017=1025.358,-91.510,410.879,166.650,46.328,158.453
C09018=1025.352,-91.760,410.889,166.646,46.331,158.453
C09019=1025.346,-92.009,410.899,166.644,46.333,158.453
C09020=1025.340,-92.259,410.909,166.641,46.336,158.454
C09021=1025.334,-92.509,410.919,166.637,46.339,158.453
C09022=1025.329,-92.758,410.929,166.635,46.341,158.454
C09023=1025.323,-93.008,410.938,166.631,46.345,158.454
C09024=1025.317,-93.258,410.948,166.628,46.348,158.454
C09025=1025.312,-93.508,410.958,166.626,46.350,158.454
C09026=1025.305,-93.758,410.968,166.622,46.353,158.454
C09027=1025.301,-94.007,410.977,166.620,46.355,158.454
C09028=1025.294,-94.257,410.987,166.617,46.359,158.455
C09029=1025.289,-94.507,410.998,166.613,46.361,158.455
C09030=1025.283,-94.756,411.007,166.611,46.364,158.455
C09031=1025.278,-95.006,411.017,166.608,46.367,158.455
C09032=1025.272,-95.256,411.027,166.604,46.369,158.455
C09033=1025.266,-95.506,411.037,166.602,46.372,158.455
C09034=1025.260,-95.756,411.046,166.598,46.375,158.455
C09035=1025.255,-96.005,411.056,166.596,46.378,158.455
C09036=1025.249,-96.255,411.066,166.593,46.380,158.455
C09037=1025.243,-96.505,411.076,166.589,46.383,158.456
C09038=1025.238,-96.754,411.085,166.587,46.386,158.456
C09039=1025.232,-97.004,411.095,166.584,46.389,158.456
C09040=1025.226,-97.254,411.105,166.580,46.391,158.456
C09041=1025.220,-97.504,411.114,166.578,46.394,158.456
C09042=1025.215,-97.753,411.124,166.575,46.397,158.456
C09043=1025.209,-98.003,411.133,166.571,46.400,158.456
C09044=1025.203,-98.253,411.143,166.569,46.403,158.457
C09045=1025.198,-98.502,411.152,166.566,46.406,158.457
C09046=1025.192,-98.752,411.162,166.562,46.408,158.457
C09047=1025.186,-99.002,411.172,166.560,46.411,158.457
C09048=1025.181,-99.251,411.181,166.557,46.414,158.457
C09049=1025.175,-99.502,411.190,166.553,46.417,158.457
C09050=1025.168,-99.752,411.199,166.551,46.420,158.457
C09051=1025.164,-100.001,411.209,166.548,46.423,158.458
C09052=1025.157,-100.251,411.219,166.544,46.426,158.458
C09053=1025.152,-100.501,411.227,166.541,46.429,158.458
C09054=1025.145,-100.786,411.239,166.538,46.432,158.458
C09055=1025.138,-101.073,411.250,166.535,46.435,158.458
C09056=1025.132,-101.359,411.259,166.532,46.439,158.458
C09057=1025.125,-101.644,411.271,166.527,46.442,158.458
C09058=1025.119,-101.894,411.280,166.525,46.445,158.459
C09059=1025.113,-102.144,411.289,166.522,46.448,158.459
C09060=1025.108,-102.394,411.299,166.518,46.451,158.459
C09061=1025.102,-102.644,411.308,166.516,46.454,158.459
C09062=1025.097,-102.893,411.317,166.512,46.456,158.459
C09063=1025.091,-103.143,411.326,166.509,46.459,158.459
C09064=1025.085,-103.393,411.335,166.507,46.462,158.460
C09065=1025.079,-103.642,411.345,166.504,46.465,158.460
C09066=1025.074,-103.892,411.355,166.500,46.468,158.460
C09067=1025.069,-104.142,411.363,166.498,46.471,158.460
C09068=1025.062,-104.392,411.373,166.495,46.474,158.460
C09069=1025.057,-104.641,411.382,166.491,46.477,158.460
C09070=1025.051,-104.892,411.391,166.488,46.480,158.460
C09071=1025.045,-105.141,411.400,166.486,46.482,158.460
C09072=1025.040,-105.391,411.409,166.482,46.485,158.461
C09073=1025.035,-105.640,411.419,166.479,46.488,158.461
C09074=1025.029,-105.890,411.428,166.477,46.491,158.461
C09075=1025.023,-106.141,411.437,166.473,46.494,158.461
C09076=1025.017,-106.390,411.446,166.470,46.497,158.461
C09077=1025.011,-106.640,411.455,166.468,46.500,158.461
C09078=1025.006,-106.889,411.464,166.465,46.503,158.462
C09079=1025.000,-107.140,411.473,166.461,46.506,158.462
C09080=1024.994,-107.389,411.482,166.458,46.509,158.462
C09081=1024.988,-107.639,411.491,166.455,46.511,158.462
C09082=1024.983,-107.888,411.500,166.452,46.514,158.462
C09083=1024.977,-108.139,411.509,166.449,46.517,158.462
C09084=1024.971,-108.388,411.518,166.447,46.520,158.462
C09085=1024.966,-108.638,411.527,166.443,46.523,158.462
C09086=1024.960,-108.887,411.537,166.440,46.526,158.463
C09087=1024.955,-109.137,411.545,166.437,46.529,158.463
C09088=1024.949,-109.387,411.554,166.434,46.532,158.463
C09089=1024.943,-109.637,411.563,166.431,46.535,158.463
C09090=1024.937,-109.887,411.572,166.428,46.538,158.463
C09091=1024.932,-110.136,411.581,166.425,46.541,158.463
C09092=1024.926,-110.386,411.590,166.422,46.544,158.464
C09093=1024.921,-110.636,411.598,166.419,46.547,158.464
C09094=1024.915,-110.886,411.608,166.416,46.550,158.464
C09095=1024.909,-111.136,411.617,166.413,46.553,158.464
C09096=1024.904,-111.385,411.625,166.410,46.556,158.464
C09097=1024.898,-111.635,411.635,166.407,46.559,158.464
C09098=1024.893,-111.885,411.643,166.404,46.562,158.464
C09099=1024.887,-112.135,411.652,166.401,46.565,158.465
C09100=1024.880,-112.384,411.661,166.398,46.568,158.465
C09101=1024.875,-112.634,411.669,166.395,46.571,158.465
C09102=1024.869,-112.884,411.678,166.391,46.574,158.465
C09103=1024.864,-113.133,411.687,166.389,46.577,158.465
C09104=1024.858,-113.383,411.696,166.386,46.580,158.465
C09105=1024.853,-113.633,411.704,166.383,46.583,158.465
C09106=1024.847,-113.883,411.713,166.380,46.586,158.466
C09107=1024.841,-114.133,411.722,166.377,46.589,158.466
C09108=1024.836,-114.383,411.731,166.374,46.592,158.466
